Yaskawa INFORM job: aprem3TRJ1.JBI

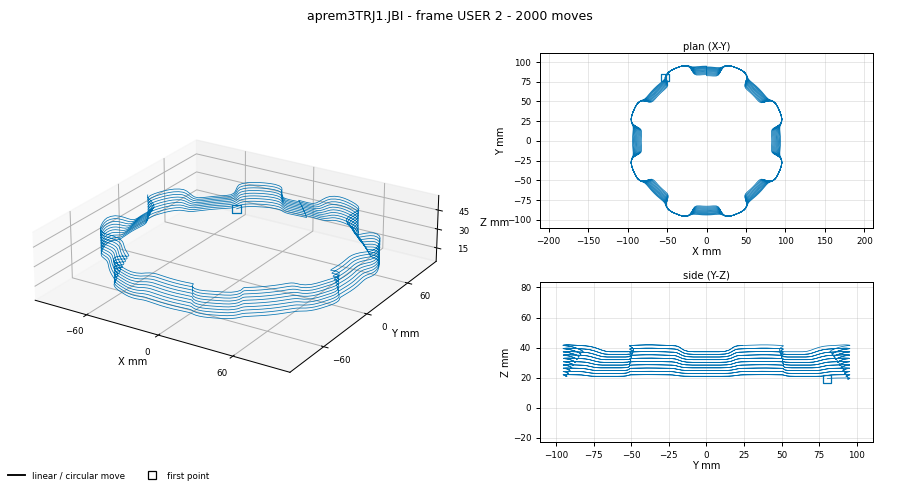
[picture p0: tool path of aprem3TRJ1.JBI in frame USER 2, 2000 of 2000 moves have a stored position in this frame; points joined in program order, loops and branches not executed]
/JOB
//NAME aprem3TRJ1
///FOLDERNAME DEMO
//POS
///NPOS 2000,0,2000,0,0,0
///USER 2
///TOOL 7
///POSTYPE USER
///RECTAN
///RCONF 1,0,0,0,0,0,0,0,0,0,0,0,0,0,0,0,0,0,0,0,0,0,0,0
C00000=-52.755,80.388,19.309,-171.7434,14.7955,-3566.7249
C00001=-51.961,81.931,19.493,-175.4363,10.0997,-3567.6170
C00002=-51.163,83.502,19.627,-176.4604,6.1368,-3568.5035
C00003=-49.917,85.194,19.692,-177.1673,3.1412,-3569.6330
C00004=-47.874,87.106,19.726,-178.6253,1.1228,-3571.2065
C00005=-45.272,88.975,19.753,-179.7684,0.1462,-3573.0322
C00006=-42.449,90.515,19.780,-179.9313,0.0331,-3574.8747
C00007=-39.659,91.796,19.798,-179.9923,0.0034,-3576.6340
C00008=-36.867,92.953,19.798,-179.9922,0.0031,-3578.3657
C00009=-33.988,94.020,19.780,-179.9280,0.0252,-3580.1252
C00010=-30.903,94.927,19.753,-179.7329,0.0604,-3581.9676
C00011=-27.741,95.446,19.726,-178.2343,0.1783,-3583.7937
C00012=-24.945,95.538,19.692,-175.7796,-0.2187,-3585.3667
C00013=-22.867,95.222,19.627,-173.1704,-1.8493,-3586.4965
C00014=-21.192,94.676,19.493,-169.6633,-3.9762,-3587.3831
C00015=-19.540,94.146,19.309,-163.8609,-4.8105,-3588.2747
C00016=-17.528,93.824,19.120,-157.6135,-2.4711,-3589.4181
C00017=-14.592,93.857,18.976,-154.0584,1.6115,-3591.1629
C00018=-10.190,94.262,18.917,-153.0799,2.7335,-3593.8301
C00019=-5.317,94.652,18.914,-152.9496,1.6756,-3596.7848
C00020=0.000,94.804,18.916,-152.9230,0.0002,-3600.0000
C00021=0.000,93.772,20.859,-151.1709,0.0003,-3600.0000
C00022=5.223,93.624,20.857,-151.1986,-1.7982,-3603.1930
C00023=10.031,93.243,20.860,-151.3318,-2.8339,-3606.1402
C00024=14.399,92.874,20.935,-152.4025,-1.1034,-3608.8129
C00025=17.292,92.935,21.118,-156.8210,4.1648,-3610.5402
C00026=19.271,93.399,21.361,-164.4264,6.3648,-3611.6582
C00027=20.902,94.108,21.598,-170.7334,4.7910,-3612.5225
C00028=22.556,94.852,21.773,-173.9772,2.3273,-3613.3766
C00029=24.607,95.353,21.858,-176.1452,0.4720,-3614.4702
C00030=27.423,95.407,21.902,-178.4246,-0.0969,-3616.0363
C00031=30.651,94.973,21.938,-179.8436,-0.0322,-3617.8866
C00032=33.828,94.073,21.973,-179.9356,-0.0223,-3619.7782
C00033=36.813,92.974,21.997,-179.9932,-0.0027,-3621.6011
C00034=39.712,91.773,21.997,-179.9933,-0.0029,-3623.3991
C00035=42.599,90.440,21.973,-179.9387,-0.0298,-3625.2213
C00036=45.483,88.829,21.938,-179.8667,-0.0878,-3627.1138
C00037=48.072,86.854,21.902,-178.8174,-1.0456,-3628.9637
C00038=50.025,84.825,21.858,-177.6053,-3.0607,-3630.5297
C00039=51.121,83.020,21.773,-177.3739,-5.9001,-3631.6234
C00040=51.765,81.324,21.598,-176.7889,-9.9060,-3632.4779
C00041=52.416,79.670,21.361,-173.2589,-15.4269,-3633.3415
C00042=53.488,77.942,21.118,-165.8953,-19.5067,-3634.4600
C00043=55.491,75.854,20.935,-159.0309,-19.5961,-3636.1873
C00044=58.840,73.026,20.860,-157.1386,-19.3725,-3638.8598
C00045=62.509,69.895,20.857,-157.6594,-20.1308,-3641.8071
C00046=66.307,66.307,20.859,-158.7340,-21.2663,-3645.0000
C00047=69.895,62.509,20.857,-159.8689,-22.3404,-3648.1929
C00048=73.026,58.840,20.860,-160.6271,-22.8610,-3651.1402
C00049=75.854,55.491,20.935,-160.4041,-20.9693,-3653.8127
C00050=77.942,53.488,21.118,-160.4933,-14.1047,-3655.5400
C00051=79.670,52.416,21.361,-164.5731,-6.7411,-3656.6585
C00052=81.324,51.765,21.598,-170.0940,-3.2111,-3657.5221
C00053=83.020,51.121,21.773,-174.0999,-2.6261,-3658.3766
C00054=84.825,50.025,21.858,-176.9393,-2.3947,-3659.4703
C00055=86.854,48.072,21.902,-178.9544,-1.1826,-3661.0363
C00056=88.829,45.483,21.938,-179.9122,-0.1333,-3662.8862
C00057=90.440,42.599,21.973,-179.9702,-0.0613,-3664.7787
C00058=91.773,39.712,21.997,-179.9971,-0.0067,-3666.6009
C00059=92.974,36.813,21.997,-179.9973,-0.0068,-3668.3989
C00060=94.073,33.828,21.973,-179.9777,-0.0644,-3670.2218
C00061=94.973,30.651,21.938,-179.9678,-0.1564,-3672.1134
C00062=95.407,27.423,21.902,-179.9031,-1.5754,-3673.9637
C00063=95.353,24.607,21.858,179.5280,-3.8548,-3675.5298
C00064=94.852,22.556,21.773,177.6727,-6.0228,-3676.6234
C00065=94.108,20.902,21.598,175.2090,-9.2666,-3677.4775
C00066=93.399,19.271,21.361,173.6352,-15.5736,-3678.3418
C00067=92.935,17.292,21.118,175.8352,-23.1790,-3679.4598
C00068=92.874,14.399,20.935,-178.8966,-27.5975,-3681.1871
C00069=93.243,10.031,20.860,-177.1661,-28.6682,-3683.8598
C00070=93.624,5.223,20.857,-178.2018,-28.8014,-3686.8070
C00071=93.772,0.000,20.859,179.9997,-28.8291,-3690.0000
C00072=93.624,-5.223,20.857,178.2021,-28.8014,-3693.1930
C00073=93.243,-10.031,20.860,177.1667,-28.6682,-3696.1402
C00074=92.875,-14.399,20.935,178.8963,-27.5974,-3698.8128
C00075=92.935,-17.292,21.118,-175.8352,-23.1790,-3700.5402
C00076=93.399,-19.271,21.361,-173.6352,-15.5736,-3701.6582
C00077=94.108,-20.902,21.598,-175.2090,-9.2666,-3702.5225
C00078=94.852,-22.556,21.773,-177.6727,-6.0228,-3703.3766
C00079=95.353,-24.607,21.858,-179.5280,-3.8548,-3704.4702
C00080=95.407,-27.423,21.902,179.9031,-1.5754,-3706.0363
C00081=94.973,-30.651,21.938,179.9678,-0.1564,-3707.8866
C00082=94.073,-33.828,21.973,179.9777,-0.0644,-3709.7782
C00083=92.974,-36.813,21.997,179.9973,-0.0068,-3711.6011
C00084=91.773,-39.712,21.997,179.9971,-0.0067,-3713.3991
C00085=90.440,-42.599,21.973,179.9702,-0.0613,-3715.2213
C00086=88.829,-45.483,21.938,179.9122,-0.1333,-3717.1138
C00087=86.854,-48.072,21.902,178.9544,-1.1826,-3718.9637
C00088=84.825,-50.025,21.858,176.9393,-2.3947,-3720.5297
C00089=83.020,-51.121,21.773,174.0999,-2.6261,-3721.6234
C00090=81.324,-51.765,21.598,170.0940,-3.2111,-3722.4779
C00091=79.670,-52.416,21.361,164.5731,-6.7411,-3723.3415
C00092=77.942,-53.488,21.118,160.4933,-14.1047,-3724.4600
C00093=75.854,-55.491,20.935,160.4039,-20.9691,-3726.1873
C00094=73.026,-58.840,20.860,160.6275,-22.8614,-3728.8598
C00095=69.895,-62.509,20.857,159.8692,-22.3406,-3731.8071
C00096=66.307,-66.307,20.859,158.7337,-21.2660,-3735.0000
C00097=62.509,-69.895,20.857,157.6596,-20.1311,-3738.1929
C00098=58.840,-73.026,20.860,157.1390,-19.3729,-3741.1402
C00099=55.491,-75.854,20.935,159.0307,-19.5959,-3743.8127
C00100=53.488,-77.942,21.118,165.8953,-19.5067,-3745.5400
C00101=52.416,-79.670,21.361,173.2589,-15.4269,-3746.6585
C00102=51.765,-81.324,21.598,176.7889,-9.9060,-3747.5221
C00103=51.121,-83.020,21.773,177.3739,-5.9001,-3748.3766
C00104=50.025,-84.825,21.858,177.6053,-3.0607,-3749.4703
C00105=48.072,-86.854,21.902,178.8174,-1.0456,-3751.0363
C00106=45.483,-88.829,21.938,179.8667,-0.0878,-3752.8862
C00107=42.599,-90.440,21.973,179.9387,-0.0298,-3754.7787
C00108=39.712,-91.773,21.997,179.9933,-0.0029,-3756.6009
C00109=36.813,-92.974,21.997,179.9932,-0.0027,-3758.3989
C00110=33.828,-94.073,21.973,179.9356,-0.0223,-3760.2218
C00111=30.651,-94.973,21.938,179.8436,-0.0322,-3762.1134
C00112=27.423,-95.407,21.902,178.4246,-0.0969,-3763.9637
C00113=24.607,-95.353,21.858,176.1452,0.4720,-3765.5298
C00114=22.556,-94.852,21.773,173.9772,2.3273,-3766.6234
C00115=20.902,-94.108,21.598,170.7334,4.7910,-3767.4775
C00116=19.271,-93.399,21.361,164.4264,6.3648,-3768.3418
C00117=17.292,-92.935,21.118,156.8210,4.1648,-3769.4598
C00118=14.399,-92.874,20.935,152.4025,-1.1034,-3771.1871
C00119=10.031,-93.243,20.860,151.3318,-2.8339,-3773.8598
C00120=5.223,-93.624,20.857,151.1986,-1.7982,-3776.8070
C00121=0.000,-93.772,20.859,151.1709,0.0003,-3780.0000
C00122=0.000,-93.772,20.859,151.1709,0.0003,-3780.0000
C00123=-5.223,-93.624,20.857,151.1986,1.7979,-3783.1930
C00124=-10.031,-93.243,20.860,151.3318,2.8333,-3786.1402
C00125=-14.399,-92.875,20.935,152.4026,1.1037,-3788.8128
C00126=-17.292,-92.935,21.118,156.8210,-4.1648,-3790.5402
C00127=-19.271,-93.399,21.361,164.4264,-6.3648,-3791.6582
C00128=-20.902,-94.108,21.598,170.7334,-4.7910,-3792.5225
C00129=-22.556,-94.852,21.773,173.9772,-2.3273,-3793.3766
C00130=-24.607,-95.353,21.858,176.1452,-0.4720,-3794.4702
C00131=-27.423,-95.407,21.902,178.4246,0.0969,-3796.0363
C00132=-30.651,-94.973,21.938,179.8436,0.0322,-3797.8866
C00133=-33.828,-94.073,21.973,179.9356,0.0223,-3799.7782
C00134=-36.813,-92.974,21.997,179.9932,0.0027,-3801.6011
C00135=-39.712,-91.773,21.997,179.9933,0.0029,-3803.3991
C00136=-42.599,-90.440,21.973,179.9387,0.0298,-3805.2213
C00137=-45.483,-88.829,21.938,179.8667,0.0878,-3807.1138
C00138=-48.072,-86.854,21.902,178.8174,1.0456,-3808.9637
C00139=-50.025,-84.825,21.858,177.6053,3.0607,-3810.5297
C00140=-51.121,-83.020,21.773,177.3739,5.9001,-3811.6234
C00141=-51.765,-81.324,21.598,176.7889,9.9060,-3812.4779
C00142=-52.416,-79.670,21.361,173.2589,15.4269,-3813.3415
C00143=-53.488,-77.942,21.118,165.8953,19.5067,-3814.4600
C00144=-55.491,-75.854,20.935,159.0309,19.5961,-3816.1873
C00145=-58.840,-73.026,20.860,157.1386,19.3725,-3818.8598
C00146=-62.509,-69.895,20.857,157.6594,20.1308,-3821.8071
C00147=-66.307,-66.307,20.859,158.7340,21.2663,-3825.0000
C00148=-69.895,-62.509,20.857,159.8689,22.3404,-3828.1929
C00149=-73.026,-58.840,20.860,160.6271,22.8610,-3831.1402
C00150=-75.854,-55.491,20.935,160.4041,20.9693,-3833.8127
C00151=-77.942,-53.488,21.118,160.4933,14.1047,-3835.5400
C00152=-79.670,-52.416,21.361,164.5731,6.7411,-3836.6585
C00153=-81.324,-51.765,21.598,170.0940,3.2111,-3837.5221
C00154=-83.020,-51.121,21.773,174.0999,2.6261,-3838.3766
C00155=-84.825,-50.025,21.858,176.9393,2.3947,-3839.4703
C00156=-86.854,-48.072,21.902,178.9544,1.1826,-3841.0363
C00157=-88.829,-45.483,21.938,179.9122,0.1333,-3842.8862
C00158=-90.440,-42.599,21.973,179.9702,0.0613,-3844.7787
C00159=-91.773,-39.712,21.997,179.9971,0.0067,-3846.6009
C00160=-92.974,-36.813,21.997,179.9973,0.0068,-3848.3989
C00161=-94.073,-33.828,21.973,179.9777,0.0644,-3850.2218
C00162=-94.973,-30.651,21.938,179.9678,0.1564,-3852.1134
C00163=-95.407,-27.423,21.902,179.9031,1.5754,-3853.9637
C00164=-95.353,-24.607,21.858,-179.5280,3.8548,-3855.5298
C00165=-94.852,-22.556,21.773,-177.6727,6.0228,-3856.6234
C00166=-94.108,-20.902,21.598,-175.2090,9.2666,-3857.4775
C00167=-93.399,-19.271,21.361,-173.6352,15.5736,-3858.3418
C00168=-92.935,-17.292,21.118,-175.8352,23.1790,-3859.4598
C00169=-92.874,-14.399,20.935,178.8966,27.5975,-3861.1871
C00170=-93.243,-10.031,20.860,177.1661,28.6682,-3863.8598
C00171=-93.624,-5.223,20.857,178.2018,28.8014,-3866.8070
C00172=-93.772,0.000,20.859,-179.9997,28.8291,-3870.0000
C00173=-93.624,5.223,20.857,-178.2021,28.8014,-3873.1930
C00174=-93.243,10.031,20.860,-177.1667,28.6682,-3876.1402
C00175=-92.875,14.399,20.935,-178.8963,27.5974,-3878.8128
C00176=-92.935,17.292,21.118,175.8352,23.1790,-3880.5402
C00177=-93.399,19.271,21.361,173.6352,15.5736,-3881.6582
C00178=-94.108,20.902,21.598,175.2090,9.2666,-3882.5225
C00179=-94.852,22.556,21.773,177.6727,6.0228,-3883.3766
C00180=-95.353,24.607,21.858,179.5280,3.8548,-3884.4702
C00181=-95.407,27.423,21.902,-179.9031,1.5754,-3886.0363
C00182=-94.973,30.651,21.938,-179.9678,0.1564,-3887.8866
C00183=-94.073,33.828,21.973,-179.9777,0.0644,-3889.7782
C00184=-92.974,36.813,21.997,-179.9973,0.0068,-3891.6011
C00185=-91.773,39.712,21.997,-179.9971,0.0067,-3893.3991
C00186=-90.440,42.599,21.973,-179.9702,0.0613,-3895.2213
C00187=-88.829,45.483,21.938,-179.9122,0.1333,-3897.1138
C00188=-86.854,48.072,21.902,-178.9544,1.1826,-3898.9637
C00189=-84.825,50.025,21.858,-176.9393,2.3947,-3900.5297
C00190=-83.020,51.121,21.773,-174.0999,2.6261,-3901.6234
C00191=-81.324,51.765,21.598,-170.0940,3.2111,-3902.4779
C00192=-79.670,52.416,21.361,-164.5731,6.7411,-3903.3415
C00193=-77.942,53.488,21.118,-160.4933,14.1047,-3904.4600
C00194=-75.854,55.491,20.935,-160.4039,20.9691,-3906.1873
C00195=-73.026,58.840,20.860,-160.6275,22.8614,-3908.8598
C00196=-69.895,62.509,20.857,-159.8692,22.3406,-3911.8071
C00197=-66.307,66.307,20.859,-158.7337,21.2660,-3915.0000
C00198=-62.509,69.895,20.857,-157.6596,20.1311,-3918.1929
C00199=-58.840,73.026,20.860,-157.1390,19.3729,-3921.1402
C00200=-55.491,75.854,20.935,-159.0307,19.5959,-3923.8127
C00201=-53.488,77.942,21.118,-165.8953,19.5067,-3925.5400
C00202=-52.416,79.670,21.361,-173.2589,15.4269,-3926.6585
C00203=-51.765,81.324,21.598,-176.7889,9.9060,-3927.5221
C00204=-51.121,83.020,21.773,-177.3739,5.9001,-3928.3766
C00205=-50.025,84.825,21.858,-177.6053,3.0607,-3929.4703
C00206=-48.072,86.854,21.902,-178.8174,1.0456,-3931.0363
C00207=-45.483,88.829,21.938,-179.8667,0.0878,-3932.8862
C00208=-42.599,90.440,21.973,-179.9387,0.0298,-3934.7787
C00209=-39.712,91.773,21.997,-179.9933,0.0029,-3936.6009
C00210=-36.813,92.974,21.997,-179.9932,0.0027,-3938.3989
C00211=-33.828,94.073,21.973,-179.9356,0.0223,-3940.2218
C00212=-30.651,94.973,21.938,-179.8436,0.0322,-3942.1134
C00213=-27.423,95.407,21.902,-178.4246,0.0969,-3943.9637
C00214=-24.607,95.353,21.858,-176.1452,-0.4720,-3945.5298
C00215=-22.556,94.852,21.773,-173.9772,-2.3273,-3946.6234
C00216=-20.902,94.108,21.598,-170.7334,-4.7910,-3947.4775
C00217=-19.271,93.399,21.361,-164.4264,-6.3648,-3948.3418
C00218=-17.292,92.935,21.118,-156.8210,-4.1648,-3949.4598
C00219=-14.399,92.875,20.935,-152.4026,1.1037,-3951.1872
C00220=-10.031,93.243,20.860,-151.3318,2.8333,-3953.8598
C00221=-5.223,93.624,20.857,-151.1986,1.7979,-3956.8070
C00222=0.000,93.772,20.859,-151.1709,0.0003,-3960.0000
C00223=0.000,92.684,22.771,-149.6099,0.0003,-3960.0000
C00224=5.124,92.540,22.769,-149.6384,-1.9089,-3963.1693
C00225=9.864,92.169,22.773,-149.7740,-2.8935,-3966.1086
C00226=14.194,91.838,22.865,-150.9609,-0.4562,-3968.7858
C00227=17.042,91.994,23.091,-156.4950,5.9927,-3970.4951
C00228=18.986,92.606,23.393,-165.5257,7.6266,-3971.5862
C00229=20.592,93.503,23.691,-172.1237,5.1935,-3972.4199
C00230=22.223,94.456,23.912,-175.0607,2.5303,-3973.2394
C00231=24.245,95.156,24.019,-176.7061,0.6541,-3974.2944
C00232=27.082,95.366,24.075,-178.6926,-0.0269,-3975.8535
C00233=30.380,95.022,24.120,-179.9786,-0.0040,-3977.7299
C00234=33.658,94.129,24.166,-179.9455,-0.0187,-3979.6757
C00235=36.755,92.996,24.196,-179.9945,-0.0022,-3981.5655
C00236=39.769,91.748,24.196,-179.9946,-0.0024,-3983.4348
C00237=42.760,90.359,24.166,-179.9482,-0.0253,-3985.3246
C00238=45.709,88.673,24.120,-179.9821,-0.0123,-3987.2701
C00239=48.284,86.584,24.075,-179.0565,-0.9056,-3989.1464
C00240=50.142,84.429,24.019,-178.1315,-2.7920,-3990.7059
C00241=51.076,82.504,23.912,-178.2896,-5.2767,-3991.7605
C00242=51.556,80.678,23.691,-178.0785,-9.2071,-3992.5800
C00243=52.057,78.907,23.393,-174.9794,-15.4942,-3993.4139
C00244=52.999,77.101,23.091,-166.8676,-20.8949,-3994.5045
C00245=54.903,74.976,22.865,-158.2868,-21.1542,-3996.2144
C00246=58.198,72.148,22.773,-155.8812,-20.6181,-3998.8913
C00247=61.813,69.059,22.769,-156.3569,-21.3383,-4001.8309
C00248=65.538,65.538,22.771,-157.4767,-22.5237,-4005.0000
C00249=69.059,61.813,22.769,-158.6615,-23.6429,-4008.1691
C00250=72.148,58.198,22.773,-159.3815,-24.1184,-4011.1087
C00251=74.976,54.903,22.865,-158.8460,-21.7135,-4013.7856
C00252=77.101,52.999,23.091,-159.1051,-13.1324,-4015.4955
C00253=78.907,52.057,23.393,-164.5058,-5.0206,-4016.5861
C00254=80.678,51.556,23.691,-170.7929,-1.9215,-4017.4200
C00255=82.504,51.076,23.912,-174.7233,-1.7104,-4018.2395
C00256=84.429,50.142,24.019,-177.2080,-1.8685,-4019.2941
C00257=86.584,48.284,24.075,-179.0944,-0.9435,-4020.8536
C00258=88.673,45.709,24.120,-179.9877,-0.0179,-4022.7299
C00259=90.359,42.760,24.166,-179.9747,-0.0518,-4024.6754
C00260=91.748,39.769,24.196,-179.9976,-0.0054,-4026.5652
C00261=92.996,36.755,24.196,-179.9978,-0.0055,-4028.4345
C00262=94.129,33.658,24.166,-179.9813,-0.0545,-4030.3243
C00263=95.022,30.380,24.120,-179.9960,-0.0214,-4032.2701
C00264=95.366,27.082,24.075,-179.9731,-1.3074,-4034.1465
C00265=95.156,24.245,24.019,179.3459,-3.2939,-4035.7056
C00266=94.456,22.223,23.912,177.4697,-4.9393,-4036.7606
C00267=93.503,20.592,23.691,174.8065,-7.8763,-4037.5801
C00268=92.606,18.986,23.393,172.3734,-14.4743,-4038.4138
C00269=91.994,17.042,23.091,174.0073,-23.5050,-4039.5049
C00270=91.838,14.194,22.865,-179.5438,-29.0391,-4041.2142
C00271=92.169,9.864,22.773,-177.1065,-30.2260,-4043.8914
C00272=92.540,5.124,22.769,-178.0911,-30.3616,-4046.8307
C00273=92.684,0.000,22.771,179.9997,-30.3901,-4050.0000
C00274=92.540,-5.124,22.769,178.0916,-30.3616,-4053.1693
C00275=92.169,-9.864,22.773,177.1071,-30.2260,-4056.1086
C00276=91.838,-14.194,22.865,179.5434,-29.0390,-4058.7858
C00277=91.994,-17.042,23.091,-174.0073,-23.5050,-4060.4951
C00278=92.606,-18.986,23.393,-172.3734,-14.4743,-4061.5862
C00279=93.503,-20.592,23.691,-174.8065,-7.8763,-4062.4199
C00280=94.456,-22.223,23.912,-177.4697,-4.9393,-4063.2394
C00281=95.156,-24.245,24.019,-179.3459,-3.2939,-4064.2944
C00282=95.366,-27.082,24.075,179.9731,-1.3074,-4065.8535
C00283=95.022,-30.380,24.120,179.9960,-0.0214,-4067.7299
C00284=94.129,-33.658,24.166,179.9813,-0.0545,-4069.6757
C00285=92.996,-36.755,24.196,179.9978,-0.0055,-4071.5655
C00286=91.748,-39.769,24.196,179.9976,-0.0054,-4073.4348
C00287=90.359,-42.760,24.166,179.9747,-0.0518,-4075.3246
C00288=88.673,-45.709,24.120,179.9877,-0.0179,-4077.2701
C00289=86.584,-48.284,24.075,179.0944,-0.9435,-4079.1464
C00290=84.429,-50.142,24.019,177.2080,-1.8685,-4080.7059
C00291=82.504,-51.076,23.912,174.7233,-1.7104,-4081.7605
C00292=80.678,-51.556,23.691,170.7929,-1.9215,-4082.5800
C00293=78.907,-52.057,23.393,164.5058,-5.0206,-4083.4139
C00294=77.101,-52.999,23.091,159.1051,-13.1324,-4084.5045
C00295=74.976,-54.903,22.865,158.8458,-21.7132,-4086.2144
C00296=72.148,-58.198,22.773,159.3819,-24.1188,-4088.8913
C00297=69.059,-61.813,22.769,158.6617,-23.6431,-4091.8309
C00298=65.538,-65.538,22.771,157.4763,-22.5233,-4095.0000
C00299=61.813,-69.059,22.769,156.3571,-21.3385,-4098.1691
C00300=58.198,-72.148,22.773,155.8816,-20.6185,-4101.1087
C00301=54.903,-74.976,22.865,158.2865,-21.1540,-4103.7856
C00302=52.999,-77.101,23.091,166.8676,-20.8949,-4105.4955
C00303=52.057,-78.907,23.393,174.9794,-15.4942,-4106.5861
C00304=51.556,-80.678,23.691,178.0785,-9.2071,-4107.4200
C00305=51.076,-82.504,23.912,178.2896,-5.2767,-4108.2395
C00306=50.142,-84.429,24.019,178.1315,-2.7920,-4109.2941
C00307=48.284,-86.584,24.075,179.0565,-0.9056,-4110.8536
C00308=45.709,-88.673,24.120,179.9821,-0.0123,-4112.7299
C00309=42.760,-90.359,24.166,179.9482,-0.0253,-4114.6754
C00310=39.769,-91.748,24.196,179.9946,-0.0024,-4116.5652
C00311=36.755,-92.996,24.196,179.9945,-0.0022,-4118.4345
C00312=33.658,-94.129,24.166,179.9455,-0.0187,-4120.3243
C00313=30.380,-95.022,24.120,179.9786,-0.0040,-4122.2701
C00314=27.082,-95.366,24.075,178.6926,-0.0269,-4124.1465
C00315=24.245,-95.156,24.019,176.7061,0.6541,-4125.7056
C00316=22.223,-94.456,23.912,175.0607,2.5303,-4126.7606
C00317=20.592,-93.503,23.691,172.1237,5.1935,-4127.5801
C00318=18.986,-92.606,23.393,165.5257,7.6266,-4128.4138
C00319=17.042,-91.994,23.091,156.4950,5.9927,-4129.5049
C00320=14.194,-91.838,22.865,150.9609,-0.4562,-4131.2142
C00321=9.864,-92.169,22.773,149.7740,-2.8935,-4133.8914
C00322=5.124,-92.540,22.769,149.6384,-1.9089,-4136.8307
C00323=0.000,-92.684,22.771,149.6099,0.0003,-4140.0000
C00324=0.000,-92.684,22.771,149.6099,0.0003,-4140.0000
C00325=-5.124,-92.540,22.769,149.6384,1.9084,-4143.1693
C00326=-9.864,-92.169,22.773,149.7740,2.8929,-4146.1086
C00327=-14.194,-91.838,22.865,150.9610,0.4566,-4148.7858
C00328=-17.042,-91.994,23.091,156.4950,-5.9927,-4150.4951
C00329=-18.986,-92.606,23.393,165.5257,-7.6266,-4151.5862
C00330=-20.592,-93.503,23.691,172.1237,-5.1935,-4152.4199
C00331=-22.223,-94.456,23.912,175.0607,-2.5303,-4153.2394
C00332=-24.245,-95.156,24.019,176.7061,-0.6541,-4154.2944
C00333=-27.082,-95.366,24.075,178.6926,0.0269,-4155.8535
C00334=-30.380,-95.022,24.120,179.9786,0.0040,-4157.7299
C00335=-33.658,-94.129,24.166,179.9455,0.0187,-4159.6757
C00336=-36.755,-92.996,24.196,179.9945,0.0022,-4161.5655
C00337=-39.769,-91.748,24.196,179.9946,0.0024,-4163.4348
C00338=-42.760,-90.359,24.166,179.9482,0.0253,-4165.3246
C00339=-45.709,-88.673,24.120,179.9821,0.0123,-4167.2701
C00340=-48.284,-86.584,24.075,179.0565,0.9056,-4169.1464
C00341=-50.142,-84.429,24.019,178.1315,2.7920,-4170.7059
C00342=-51.076,-82.504,23.912,178.2896,5.2767,-4171.7605
C00343=-51.556,-80.678,23.691,178.0785,9.2071,-4172.5800
C00344=-52.057,-78.907,23.393,174.9794,15.4942,-4173.4139
C00345=-52.999,-77.101,23.091,166.8676,20.8949,-4174.5045
C00346=-54.903,-74.976,22.865,158.2868,21.1542,-4176.2144
C00347=-58.198,-72.148,22.773,155.8812,20.6181,-4178.8913
C00348=-61.813,-69.059,22.769,156.3569,21.3383,-4181.8309
C00349=-65.538,-65.538,22.771,157.4767,22.5237,-4185.0000
C00350=-69.059,-61.813,22.769,158.6615,23.6429,-4188.1691
C00351=-72.148,-58.198,22.773,159.3815,24.1184,-4191.1087
C00352=-74.976,-54.903,22.865,158.8460,21.7135,-4193.7856
C00353=-77.101,-52.999,23.091,159.1051,13.1324,-4195.4955
C00354=-78.907,-52.057,23.393,164.5058,5.0206,-4196.5861
C00355=-80.678,-51.556,23.691,170.7929,1.9215,-4197.4200
C00356=-82.504,-51.076,23.912,174.7233,1.7104,-4198.2395
C00357=-84.429,-50.142,24.019,177.2080,1.8685,-4199.2941
C00358=-86.584,-48.284,24.075,179.0944,0.9435,-4200.8536
C00359=-88.673,-45.709,24.120,179.9877,0.0179,-4202.7299
C00360=-90.359,-42.760,24.166,179.9747,0.0518,-4204.6754
C00361=-91.748,-39.769,24.196,179.9976,0.0054,-4206.5652
C00362=-92.996,-36.755,24.196,179.9978,0.0055,-4208.4345
C00363=-94.129,-33.658,24.166,179.9813,0.0545,-4210.3243
C00364=-95.022,-30.380,24.120,179.9960,0.0214,-4212.2701
C00365=-95.366,-27.082,24.075,179.9731,1.3074,-4214.1465
C00366=-95.156,-24.245,24.019,-179.3459,3.2939,-4215.7056
C00367=-94.456,-22.223,23.912,-177.4697,4.9393,-4216.7606
C00368=-93.503,-20.592,23.691,-174.8065,7.8763,-4217.5801
C00369=-92.606,-18.986,23.393,-172.3734,14.4743,-4218.4138
C00370=-91.994,-17.042,23.091,-174.0073,23.5050,-4219.5049
C00371=-91.838,-14.194,22.865,179.5438,29.0391,-4221.2142
C00372=-92.169,-9.864,22.773,177.1065,30.2260,-4223.8914
C00373=-92.540,-5.124,22.769,178.0911,30.3616,-4226.8307
C00374=-92.684,0.000,22.771,-179.9997,30.3901,-4230.0000
C00375=-92.540,5.124,22.769,-178.0916,30.3616,-4233.1693
C00376=-92.169,9.864,22.773,-177.1071,30.2260,-4236.1086
C00377=-91.838,14.194,22.865,-179.5434,29.0390,-4238.7858
C00378=-91.994,17.042,23.091,174.0073,23.5050,-4240.4951
C00379=-92.606,18.986,23.393,172.3734,14.4743,-4241.5862
C00380=-93.503,20.592,23.691,174.8065,7.8763,-4242.4199
C00381=-94.456,22.223,23.912,177.4697,4.9393,-4243.2394
C00382=-95.156,24.245,24.019,179.3459,3.2939,-4244.2944
C00383=-95.366,27.082,24.075,-179.9731,1.3074,-4245.8535
C00384=-95.022,30.380,24.120,-179.9960,0.0214,-4247.7299
C00385=-94.129,33.658,24.166,-179.9813,0.0545,-4249.6757
C00386=-92.996,36.755,24.196,-179.9978,0.0055,-4251.5655
C00387=-91.748,39.769,24.196,-179.9976,0.0054,-4253.4348
C00388=-90.359,42.760,24.166,-179.9747,0.0518,-4255.3246
C00389=-88.673,45.709,24.120,-179.9877,0.0179,-4257.2701
C00390=-86.584,48.284,24.075,-179.0944,0.9435,-4259.1464
C00391=-84.429,50.142,24.019,-177.2080,1.8685,-4260.7059
C00392=-82.504,51.076,23.912,-174.7233,1.7104,-4261.7605
C00393=-80.678,51.556,23.691,-170.7929,1.9215,-4262.5800
C00394=-78.907,52.057,23.393,-164.5058,5.0206,-4263.4139
C00395=-77.101,52.999,23.091,-159.1051,13.1324,-4264.5045
C00396=-74.976,54.903,22.865,-158.8458,21.7132,-4266.2144
C00397=-72.148,58.198,22.773,-159.3819,24.1188,-4268.8913
C00398=-69.059,61.813,22.769,-158.6617,23.6431,-4271.8309
C00399=-65.538,65.538,22.771,-157.4763,22.5233,-4275.0000
C00400=-61.813,69.059,22.769,-156.3571,21.3385,-4278.1691
C00401=-58.198,72.148,22.773,-155.8816,20.6185,-4281.1087
C00402=-54.903,74.976,22.865,-158.2865,21.1540,-4283.7856
C00403=-52.999,77.101,23.091,-166.8676,20.8949,-4285.4955
C00404=-52.057,78.907,23.393,-174.9794,15.4942,-4286.5861
C00405=-51.556,80.678,23.691,-178.0785,9.2071,-4287.4200
C00406=-51.076,82.504,23.912,-178.2896,5.2767,-4288.2395
C00407=-50.142,84.429,24.019,-178.1315,2.7920,-4289.2941
C00408=-48.284,86.584,24.075,-179.0565,0.9056,-4290.8536
C00409=-45.709,88.673,24.120,-179.9821,0.0123,-4292.7299
C00410=-42.760,90.359,24.166,-179.9482,0.0253,-4294.6754
C00411=-39.769,91.748,24.196,-179.9946,0.0024,-4296.5652
C00412=-36.755,92.996,24.196,-179.9945,0.0022,-4298.4345
C00413=-33.658,94.129,24.166,-179.9455,0.0187,-4300.3243
C00414=-30.380,95.022,24.120,-179.9786,0.0040,-4302.2701
C00415=-27.082,95.366,24.075,-178.6926,0.0269,-4304.1465
C00416=-24.245,95.156,24.019,-176.7061,-0.6541,-4305.7056
C00417=-22.223,94.456,23.912,-175.0607,-2.5303,-4306.7606
C00418=-20.592,93.503,23.691,-172.1237,-5.1935,-4307.5801
C00419=-18.986,92.606,23.393,-165.5257,-7.6266,-4308.4138
C00420=-17.042,91.994,23.091,-156.4950,-5.9927,-4309.5049
C00421=-14.194,91.838,22.865,-150.9610,0.4566,-4311.2142
C00422=-9.864,92.169,22.773,-149.7740,2.8929,-4313.8914
C00423=-5.124,92.540,22.769,-149.6384,1.9084,-4316.8307
C00424=0.000,92.684,22.771,-149.6099,0.0003,-4320.0000
C00425=0.000,91.548,24.655,-148.2220,0.0004,-4320.0000
C00426=5.020,91.408,24.652,-148.2512,-2.0082,-4323.1434
C00427=9.690,91.047,24.657,-148.3888,-2.9141,-4326.0750
C00428=13.981,90.755,24.767,-149.7234,0.3213,-4328.7577
C00429=16.781,91.008,25.041,-156.6468,7.8344,-4330.4474
C00430=18.686,91.772,25.406,-167.0189,8.4697,-4331.5089
C00431=20.265,92.865,25.771,-173.6442,5.1590,-4332.3101
C00432=21.871,94.037,26.043,-176.2884,2.4064,-4333.0930
C00433=23.861,94.948,26.175,-177.4309,0.7190,-4334.1066
C00434=26.720,95.323,26.245,-179.0289,0.0208,-4335.6587
C00435=30.093,95.074,26.301,179.8658,0.0220,-4337.5637
C00436=33.476,94.189,26.358,-179.9573,-0.0145,-4339.5659
C00437=36.693,93.020,26.395,-179.9960,-0.0016,-4341.5274
C00438=39.829,91.721,26.395,-179.9960,-0.0018,-4343.4725
C00439=42.931,90.273,26.358,-179.9596,-0.0199,-4345.4343
C00440=45.948,88.507,26.301,179.8895,0.0793,-4347.4359
C00441=48.509,86.297,26.245,-179.3280,-0.7014,-4349.3411
C00442=50.266,84.010,26.175,-178.6908,-2.3250,-4350.8935
C00443=51.029,81.959,26.043,-179.0745,-4.3225,-4351.9071
C00444=51.336,79.995,25.771,-179.1451,-8.1159,-4352.6899
C00445=51.679,78.105,25.406,-176.6973,-15.0186,-4353.4910
C00446=52.487,76.218,25.041,-168.2493,-21.9298,-4354.5530
C00447=54.287,74.059,24.767,-157.7629,-22.6253,-4356.2423
C00448=57.528,71.231,24.657,-154.7702,-21.7624,-4358.9252
C00449=61.085,68.184,24.652,-155.1868,-22.4287,-4361.8567
C00450=64.734,64.734,24.655,-156.3444,-23.6560,-4365.0000
C00451=68.184,61.085,24.652,-157.5710,-24.8129,-4368.1433
C00452=71.231,57.528,24.657,-158.2372,-25.2293,-4371.0748
C00453=74.059,54.287,24.767,-157.3750,-22.2374,-4373.7577
C00454=76.218,52.487,25.041,-158.0702,-11.7507,-4375.4470
C00455=78.105,51.679,25.406,-164.9814,-3.3027,-4376.5090
C00456=79.995,51.336,25.771,-171.8841,-0.8549,-4377.3101
C00457=81.959,51.029,26.043,-175.6775,-0.9255,-4378.0929
C00458=84.010,50.266,26.175,-177.6750,-1.3092,-4379.1065
C00459=86.297,48.509,26.245,-179.2986,-0.6720,-4380.6589
C00460=88.507,45.948,26.301,179.9207,0.1105,-4382.5641
C00461=90.273,42.931,26.358,-179.9801,-0.0404,-4384.5657
C00462=91.721,39.829,26.395,-179.9982,-0.0040,-4386.5275
C00463=93.020,36.693,26.395,-179.9984,-0.0040,-4388.4726
C00464=94.189,33.476,26.358,-179.9855,-0.0427,-4390.4341
C00465=95.074,30.093,26.301,179.9780,0.1342,-4392.4363
C00466=95.323,26.720,26.245,179.9792,-0.9711,-4394.3413
C00467=94.948,23.861,26.175,179.2810,-2.5691,-4395.8934
C00468=94.037,21.871,26.043,177.5936,-3.7116,-4396.9070
C00469=92.865,20.265,25.771,174.8410,-6.3558,-4397.6899
C00470=91.772,18.686,25.406,171.5303,-12.9811,-4398.4911
C00471=91.008,16.781,25.041,172.1656,-23.3532,-4399.5526
C00472=90.755,13.981,24.767,179.6787,-30.2766,-4401.2423
C00473=91.047,9.690,24.657,-177.0859,-31.6112,-4403.9250
C00474=91.408,5.020,24.652,-177.9918,-31.7488,-4406.8566
C00475=91.548,0.000,24.655,179.9996,-31.7780,-4410.0000
C00476=91.408,-5.020,24.652,177.9923,-31.7488,-4413.1434
C00477=91.047,-9.690,24.657,177.0867,-31.6111,-4416.0750
C00478=90.755,-13.981,24.767,-179.6793,-30.2766,-4418.7577
C00479=91.008,-16.781,25.041,-172.1656,-23.3532,-4420.4474
C00480=91.772,-18.686,25.406,-171.5303,-12.9811,-4421.5089
C00481=92.865,-20.265,25.771,-174.8410,-6.3558,-4422.3101
C00482=94.037,-21.871,26.043,-177.5936,-3.7116,-4423.0930
C00483=94.948,-23.861,26.175,-179.2810,-2.5691,-4424.1066
C00484=95.323,-26.720,26.245,-179.9792,-0.9711,-4425.6587
C00485=95.074,-30.093,26.301,-179.9780,0.1342,-4427.5637
C00486=94.189,-33.476,26.358,179.9855,-0.0427,-4429.5659
C00487=93.020,-36.693,26.395,179.9984,-0.0040,-4431.5274
C00488=91.721,-39.829,26.395,179.9982,-0.0040,-4433.4725
C00489=90.273,-42.931,26.358,179.9801,-0.0404,-4435.4343
C00490=88.507,-45.948,26.301,-179.9207,0.1105,-4437.4359
C00491=86.297,-48.509,26.245,179.2986,-0.6720,-4439.3411
C00492=84.010,-50.266,26.175,177.6750,-1.3092,-4440.8935
C00493=81.959,-51.029,26.043,175.6775,-0.9255,-4441.9071
C00494=79.995,-51.336,25.771,171.8841,-0.8549,-4442.6899
C00495=78.105,-51.679,25.406,164.9814,-3.3027,-4443.4910
C00496=76.218,-52.487,25.041,158.0702,-11.7507,-4444.5530
C00497=74.059,-54.287,24.767,157.3747,-22.2371,-4446.2423
C00498=71.231,-57.528,24.657,158.2376,-25.2298,-4448.9252
C00499=68.184,-61.085,24.652,157.5713,-24.8132,-4451.8567
C00500=64.734,-64.734,24.655,156.3440,-23.6556,-4455.0000
C00501=61.085,-68.184,24.652,155.1871,-22.4290,-4458.1433
C00502=57.528,-71.231,24.657,154.7707,-21.7628,-4461.0748
C00503=54.287,-74.059,24.767,157.7626,-22.6250,-4463.7577
C00504=52.487,-76.218,25.041,168.2493,-21.9298,-4465.4470
C00505=51.679,-78.105,25.406,176.6973,-15.0186,-4466.5090
C00506=51.336,-79.995,25.771,179.1451,-8.1159,-4467.3101
C00507=51.029,-81.959,26.043,179.0745,-4.3225,-4468.0929
C00508=50.266,-84.010,26.175,178.6908,-2.3250,-4469.1065
C00509=48.509,-86.297,26.245,179.3280,-0.7014,-4470.6589
C00510=45.948,-88.507,26.301,-179.8895,0.0793,-4472.5641
C00511=42.931,-90.273,26.358,179.9596,-0.0199,-4474.5657
C00512=39.829,-91.721,26.395,179.9960,-0.0018,-4476.5275
C00513=36.693,-93.020,26.395,179.9960,-0.0016,-4478.4726
C00514=33.476,-94.189,26.358,179.9573,-0.0145,-4480.4341
C00515=30.093,-95.074,26.301,-179.8658,0.0220,-4482.4363
C00516=26.720,-95.323,26.245,179.0289,0.0208,-4484.3413
C00517=23.861,-94.948,26.175,177.4309,0.7190,-4485.8934
C00518=21.871,-94.037,26.043,176.2884,2.4064,-4486.9070
C00519=20.265,-92.865,25.771,173.6442,5.1590,-4487.6899
C00520=18.686,-91.772,25.406,167.0189,8.4697,-4488.4911
C00521=16.781,-91.008,25.041,156.6468,7.8344,-4489.5526
C00522=13.981,-90.755,24.767,149.7234,0.3213,-4491.2423
C00523=9.690,-91.047,24.657,148.3888,-2.9141,-4493.9250
C00524=5.020,-91.408,24.652,148.2512,-2.0082,-4496.8566
C00525=0.000,-91.548,24.655,148.2220,0.0004,-4500.0000
C00526=0.000,-91.548,24.655,148.2220,0.0004,-4500.0000
C00527=-5.020,-91.408,24.652,148.2512,2.0077,-4503.1434
C00528=-9.690,-91.047,24.657,148.3889,2.9133,-4506.0750
C00529=-13.981,-90.755,24.767,149.7234,-0.3207,-4508.7577
C00530=-16.781,-91.008,25.041,156.6468,-7.8344,-4510.4474
C00531=-18.686,-91.772,25.406,167.0189,-8.4697,-4511.5089
C00532=-20.265,-92.865,25.771,173.6442,-5.1590,-4512.3101
C00533=-21.871,-94.037,26.043,176.2884,-2.4064,-4513.0930
C00534=-23.861,-94.948,26.175,177.4309,-0.7190,-4514.1066
C00535=-26.720,-95.323,26.245,179.0289,-0.0208,-4515.6587
C00536=-30.093,-95.074,26.301,-179.8658,-0.0220,-4517.5637
C00537=-33.476,-94.189,26.358,179.9573,0.0145,-4519.5659
C00538=-36.693,-93.020,26.395,179.9960,0.0016,-4521.5274
C00539=-39.829,-91.721,26.395,179.9960,0.0018,-4523.4725
C00540=-42.931,-90.273,26.358,179.9596,0.0199,-4525.4343
C00541=-45.948,-88.507,26.301,-179.8895,-0.0793,-4527.4359
C00542=-48.509,-86.297,26.245,179.3280,0.7014,-4529.3411
C00543=-50.266,-84.010,26.175,178.6908,2.3250,-4530.8935
C00544=-51.029,-81.959,26.043,179.0745,4.3225,-4531.9071
C00545=-51.336,-79.995,25.771,179.1451,8.1159,-4532.6899
C00546=-51.679,-78.105,25.406,176.6973,15.0186,-4533.4910
C00547=-52.487,-76.218,25.041,168.2493,21.9298,-4534.5530
C00548=-54.287,-74.059,24.767,157.7629,22.6253,-4536.2423
C00549=-57.528,-71.231,24.657,154.7702,21.7624,-4538.9252
C00550=-61.085,-68.184,24.652,155.1868,22.4287,-4541.8567
C00551=-64.734,-64.734,24.655,156.3444,23.6560,-4545.0000
C00552=-68.184,-61.085,24.652,157.5710,24.8129,-4548.1433
C00553=-71.231,-57.528,24.657,158.2372,25.2293,-4551.0748
C00554=-74.059,-54.287,24.767,157.3750,22.2374,-4553.7577
C00555=-76.218,-52.487,25.041,158.0702,11.7507,-4555.4470
C00556=-78.105,-51.679,25.406,164.9814,3.3027,-4556.5090
C00557=-79.995,-51.336,25.771,171.8841,0.8549,-4557.3101
C00558=-81.959,-51.029,26.043,175.6775,0.9255,-4558.0929
C00559=-84.010,-50.266,26.175,177.6750,1.3092,-4559.1065
C00560=-86.297,-48.509,26.245,179.2986,0.6720,-4560.6589
C00561=-88.507,-45.948,26.301,-179.9207,-0.1105,-4562.5641
C00562=-90.273,-42.931,26.358,179.9801,0.0404,-4564.5657
C00563=-91.721,-39.829,26.395,179.9982,0.0040,-4566.5275
C00564=-93.020,-36.693,26.395,179.9984,0.0040,-4568.4726
C00565=-94.189,-33.476,26.358,179.9855,0.0427,-4570.4341
C00566=-95.074,-30.093,26.301,-179.9780,-0.1342,-4572.4363
C00567=-95.323,-26.720,26.245,-179.9792,0.9711,-4574.3413
C00568=-94.948,-23.861,26.175,-179.2810,2.5691,-4575.8934
C00569=-94.037,-21.871,26.043,-177.5936,3.7116,-4576.9070
C00570=-92.865,-20.265,25.771,-174.8410,6.3558,-4577.6899
C00571=-91.772,-18.686,25.406,-171.5303,12.9811,-4578.4911
C00572=-91.008,-16.781,25.041,-172.1656,23.3532,-4579.5526
C00573=-90.755,-13.981,24.767,-179.6787,30.2766,-4581.2423
C00574=-91.047,-9.690,24.657,177.0859,31.6112,-4583.9250
C00575=-91.408,-5.020,24.652,177.9918,31.7488,-4586.8566
C00576=-91.548,0.000,24.655,-179.9996,31.7780,-4590.0000
C00577=-91.408,5.020,24.652,-177.9923,31.7488,-4593.1434
C00578=-91.047,9.690,24.657,-177.0867,31.6111,-4596.0750
C00579=-90.755,13.981,24.767,179.6793,30.2766,-4598.7577
C00580=-91.008,16.781,25.041,172.1656,23.3532,-4600.4474
C00581=-91.772,18.686,25.406,171.5303,12.9811,-4601.5089
C00582=-92.865,20.265,25.771,174.8410,6.3558,-4602.3101
C00583=-94.037,21.871,26.043,177.5936,3.7116,-4603.0930
C00584=-94.948,23.861,26.175,179.2810,2.5691,-4604.1066
C00585=-95.323,26.720,26.245,179.9792,0.9711,-4605.6587
C00586=-95.074,30.093,26.301,179.9780,-0.1342,-4607.5637
C00587=-94.189,33.476,26.358,-179.9855,0.0427,-4609.5659
C00588=-93.020,36.693,26.395,-179.9984,0.0040,-4611.5274
C00589=-91.721,39.829,26.395,-179.9982,0.0040,-4613.4725
C00590=-90.273,42.931,26.358,-179.9801,0.0404,-4615.4343
C00591=-88.507,45.948,26.301,179.9207,-0.1105,-4617.4359
C00592=-86.297,48.509,26.245,-179.2986,0.6720,-4619.3411
C00593=-84.010,50.266,26.175,-177.6750,1.3092,-4620.8935
C00594=-81.959,51.029,26.043,-175.6775,0.9255,-4621.9071
C00595=-79.995,51.336,25.771,-171.8841,0.8549,-4622.6899
C00596=-78.105,51.679,25.406,-164.9814,3.3027,-4623.4910
C00597=-76.218,52.487,25.041,-158.0702,11.7507,-4624.5530
C00598=-74.059,54.287,24.767,-157.3747,22.2371,-4626.2423
C00599=-71.231,57.528,24.657,-158.2376,25.2298,-4628.9252
C00600=-68.184,61.085,24.652,-157.5713,24.8132,-4631.8567
C00601=-64.734,64.734,24.655,-156.3440,23.6556,-4635.0000
C00602=-61.085,68.184,24.652,-155.1871,22.4290,-4638.1433
C00603=-57.528,71.231,24.657,-154.7707,21.7628,-4641.0748
C00604=-54.287,74.059,24.767,-157.7626,22.6250,-4643.7577
C00605=-52.487,76.218,25.041,-168.2493,21.9298,-4645.4470
C00606=-51.679,78.105,25.406,-176.6973,15.0186,-4646.5090
C00607=-51.336,79.995,25.771,-179.1451,8.1159,-4647.3101
C00608=-51.029,81.959,26.043,-179.0745,4.3225,-4648.0929
C00609=-50.266,84.010,26.175,-178.6908,2.3250,-4649.1065
C00610=-48.509,86.297,26.245,-179.3280,0.7014,-4650.6589
C00611=-45.948,88.507,26.301,179.8895,-0.0793,-4652.5641
C00612=-42.931,90.273,26.358,-179.9596,0.0199,-4654.5657
C00613=-39.829,91.721,26.395,-179.9960,0.0018,-4656.5275
C00614=-36.693,93.020,26.395,-179.9960,0.0016,-4658.4726
C00615=-33.476,94.189,26.358,-179.9573,0.0145,-4660.4341
C00616=-30.093,95.074,26.301,179.8658,-0.0220,-4662.4363
C00617=-26.720,95.323,26.245,-179.0289,-0.0208,-4664.3413
C00618=-23.861,94.948,26.175,-177.4309,-0.7190,-4665.8934
C00619=-21.871,94.037,26.043,-176.2884,-2.4064,-4666.9070
C00620=-20.265,92.865,25.771,-173.6442,-5.1590,-4667.6899
C00621=-18.686,91.772,25.406,-167.0189,-8.4697,-4668.4911
C00622=-16.781,91.008,25.041,-156.6468,-7.8344,-4669.5526
C00623=-13.981,90.755,24.767,-149.7234,-0.3207,-4671.2423
C00624=-9.690,91.047,24.657,-148.3889,2.9133,-4673.9250
C00625=-5.020,91.408,24.652,-148.2512,2.0077,-4676.8566
C00626=0.000,91.548,24.655,-148.2220,0.0004,-4680.0000
C00627=0.000,90.369,26.513,-146.9909,0.0004,-4680.0000
C00628=4.912,90.233,26.509,-147.0206,-2.0967,-4683.1159
C00629=9.508,89.882,26.515,-147.1605,-2.8971,-4686.0385
C00630=13.759,89.629,26.645,-148.6809,1.2171,-4688.7274
C00631=16.509,89.983,26.968,-157.2655,9.5618,-4690.3963
C00632=18.373,90.901,27.402,-168.7365,8.8492,-4691.4267
C00633=19.923,92.196,27.838,-175.1312,4.7417,-4692.1938
C00634=21.502,93.597,28.166,-177.5251,1.9666,-4692.9380
C00635=23.458,94.728,28.327,-178.2716,0.6326,-4693.9087
C00636=26.340,95.277,28.411,-179.4215,0.0370,-4695.4538
C00637=29.791,95.129,28.479,179.6935,0.0440,-4697.3887
C00638=33.285,94.252,28.548,-179.9707,-0.0099,-4699.4506
C00639=36.628,93.045,28.594,-179.9976,-0.0009,-4701.4875
C00640=39.893,91.693,28.594,-179.9976,-0.0010,-4703.5125
C00641=43.110,90.182,28.548,-179.9723,-0.0138,-4705.5494
C00642=46.201,88.332,28.479,179.7522,0.1856,-4707.6113
C00643=48.746,85.996,28.411,-179.6171,-0.4352,-4709.5463
C00644=50.396,83.570,28.327,-179.2249,-1.6694,-4711.0916
C00645=50.979,81.387,28.166,-179.6401,-3.1392,-4712.0621
C00646=51.105,79.281,27.838,-179.9095,-6.7798,-4712.8061
C00647=51.285,77.269,27.402,-178.2394,-14.0854,-4713.5730
C00648=51.954,75.301,26.968,-169.9528,-22.5582,-4714.6038
C00649=53.649,73.106,26.645,-157.4504,-24.0022,-4716.2732
C00650=56.833,70.280,26.515,-153.7948,-22.8119,-4718.9613
C00651=60.331,67.277,26.509,-154.1393,-23.4102,-4721.8843
C00652=63.901,63.901,26.513,-155.3281,-24.6724,-4725.0000
C00653=67.277,60.331,26.509,-156.5894,-25.8604,-4728.1157
C00654=70.280,56.833,26.515,-157.1876,-26.2046,-4731.0387
C00655=73.106,53.649,26.645,-155.9981,-22.5500,-4733.7268
C00656=75.301,51.954,26.968,-157.4418,-10.0472,-4735.3962
C00657=77.269,51.285,27.402,-165.9146,-1.7606,-4736.4270
C00658=79.281,51.105,27.838,-173.2202,-0.0905,-4737.1939
C00659=81.387,50.979,28.166,-176.8608,-0.3599,-4737.9379
C00660=83.570,50.396,28.327,-178.3306,-0.7751,-4738.9084
C00661=85.996,48.746,28.411,-179.5648,-0.3829,-4740.4537
C00662=88.332,46.201,28.479,179.8144,0.2478,-4742.3887
C00663=90.182,43.110,28.548,-179.9862,-0.0277,-4744.4506
C00664=91.693,39.893,28.594,-179.9990,-0.0024,-4746.4875
C00665=93.045,36.628,28.594,-179.9991,-0.0024,-4748.5125
C00666=94.252,33.285,28.548,-179.9901,-0.0293,-4750.5494
C00667=95.129,29.791,28.479,179.9560,0.3065,-4752.6113
C00668=95.277,26.340,28.411,179.9630,-0.5785,-4754.5462
C00669=94.728,23.458,28.327,179.3674,-1.7284,-4756.0913
C00670=93.597,21.502,28.166,178.0334,-2.4749,-4757.0620
C00671=92.196,19.923,27.838,175.2583,-4.8688,-4757.8062
C00672=90.901,18.373,27.402,171.1508,-11.2635,-4758.5733
C00673=89.983,16.509,26.968,170.4382,-22.7345,-4759.6037
C00674=89.629,13.759,26.645,178.7829,-31.3191,-4761.2726
C00675=89.882,9.508,26.515,-177.1029,-32.8395,-4763.9615
C00676=90.233,4.912,26.509,-177.9033,-32.9794,-4766.8841
C00677=90.369,0.000,26.513,179.9996,-33.0091,-4770.0000
C00678=90.233,-4.912,26.509,177.9038,-32.9794,-4773.1159
C00679=89.882,-9.508,26.515,177.1039,-32.8395,-4776.0385
C00680=89.629,-13.759,26.645,-178.7835,-31.3192,-4778.7274
C00681=89.983,-16.509,26.968,-170.4382,-22.7345,-4780.3963
C00682=90.901,-18.373,27.402,-171.1508,-11.2635,-4781.4267
C00683=92.196,-19.923,27.838,-175.2583,-4.8688,-4782.1938
C00684=93.597,-21.502,28.166,-178.0334,-2.4749,-4782.9380
C00685=94.728,-23.458,28.327,-179.3674,-1.7284,-4783.9087
C00686=95.277,-26.340,28.411,-179.9630,-0.5785,-4785.4538
C00687=95.129,-29.791,28.479,-179.9560,0.3065,-4787.3887
C00688=94.252,-33.285,28.548,179.9901,-0.0293,-4789.4506
C00689=93.045,-36.628,28.594,179.9991,-0.0024,-4791.4875
C00690=91.693,-39.893,28.594,179.9990,-0.0024,-4793.5125
C00691=90.182,-43.110,28.548,179.9862,-0.0277,-4795.5494
C00692=88.332,-46.201,28.479,-179.8144,0.2478,-4797.6113
C00693=85.996,-48.746,28.411,179.5648,-0.3829,-4799.5463
C00694=83.570,-50.396,28.327,178.3306,-0.7751,-4801.0916
C00695=81.387,-50.979,28.166,176.8608,-0.3599,-4802.0621
C00696=79.281,-51.105,27.838,173.2202,-0.0905,-4802.8061
C00697=77.269,-51.285,27.402,165.9146,-1.7606,-4803.5730
C00698=75.301,-51.954,26.968,157.4418,-10.0472,-4804.6038
C00699=73.106,-53.649,26.645,155.9978,-22.5496,-4806.2732
C00700=70.280,-56.833,26.515,157.1881,-26.2052,-4808.9613
C00701=67.277,-60.331,26.509,156.5898,-25.8607,-4811.8843
C00702=63.901,-63.901,26.513,155.3276,-24.6719,-4815.0000
C00703=60.331,-67.277,26.509,154.1396,-23.4106,-4818.1157
C00704=56.833,-70.280,26.515,153.7954,-22.8124,-4821.0387
C00705=53.649,-73.106,26.645,157.4500,-24.0019,-4823.7268
C00706=51.954,-75.301,26.968,169.9528,-22.5582,-4825.3962
C00707=51.285,-77.269,27.402,178.2394,-14.0854,-4826.4270
C00708=51.105,-79.281,27.838,179.9095,-6.7798,-4827.1939
C00709=50.979,-81.387,28.166,179.6401,-3.1392,-4827.9379
C00710=50.396,-83.570,28.327,179.2249,-1.6694,-4828.9084
C00711=48.746,-85.996,28.411,179.6171,-0.4352,-4830.4537
C00712=46.201,-88.332,28.479,-179.7522,0.1856,-4832.3887
C00713=43.110,-90.182,28.548,179.9723,-0.0138,-4834.4506
C00714=39.893,-91.693,28.594,179.9976,-0.0010,-4836.4875
C00715=36.628,-93.045,28.594,179.9976,-0.0009,-4838.5125
C00716=33.285,-94.252,28.548,179.9707,-0.0099,-4840.5494
C00717=29.791,-95.129,28.479,-179.6935,0.0440,-4842.6113
C00718=26.340,-95.277,28.411,179.4215,0.0370,-4844.5462
C00719=23.458,-94.728,28.327,178.2716,0.6326,-4846.0913
C00720=21.502,-93.597,28.166,177.5251,1.9666,-4847.0620
C00721=19.923,-92.196,27.838,175.1312,4.7417,-4847.8062
C00722=18.373,-90.901,27.402,168.7365,8.8492,-4848.5733
C00723=16.509,-89.983,26.968,157.2655,9.5618,-4849.6037
C00724=13.759,-89.629,26.645,148.6809,1.2171,-4851.2726
C00725=9.508,-89.882,26.515,147.1605,-2.8971,-4853.9615
C00726=4.912,-90.233,26.509,147.0206,-2.0967,-4856.8841
C00727=0.000,-90.369,26.513,146.9909,0.0004,-4860.0000
C00728=0.000,-90.369,26.513,146.9909,0.0004,-4860.0000
C00729=-4.912,-90.233,26.509,147.0206,2.0962,-4863.1159
C00730=-9.508,-89.882,26.515,147.1605,2.8961,-4866.0385
C00731=-13.759,-89.629,26.645,148.6808,-1.2165,-4868.7274
C00732=-16.509,-89.983,26.968,157.2655,-9.5618,-4870.3963
C00733=-18.373,-90.901,27.402,168.7365,-8.8492,-4871.4267
C00734=-19.923,-92.196,27.838,175.1312,-4.7417,-4872.1938
C00735=-21.502,-93.597,28.166,177.5251,-1.9666,-4872.9380
C00736=-23.458,-94.728,28.327,178.2716,-0.6326,-4873.9087
C00737=-26.340,-95.277,28.411,179.4215,-0.0370,-4875.4538
C00738=-29.791,-95.129,28.479,-179.6935,-0.0440,-4877.3887
C00739=-33.285,-94.252,28.548,179.9707,0.0099,-4879.4506
C00740=-36.628,-93.045,28.594,179.9976,0.0009,-4881.4875
C00741=-39.893,-91.693,28.594,179.9976,0.0010,-4883.5125
C00742=-43.110,-90.182,28.548,179.9723,0.0138,-4885.5494
C00743=-46.201,-88.332,28.479,-179.7522,-0.1856,-4887.6113
C00744=-48.746,-85.996,28.411,179.6171,0.4352,-4889.5463
C00745=-50.396,-83.570,28.327,179.2249,1.6694,-4891.0916
C00746=-50.979,-81.387,28.166,179.6401,3.1392,-4892.0621
C00747=-51.105,-79.281,27.838,179.9095,6.7798,-4892.8061
C00748=-51.285,-77.269,27.402,178.2394,14.0854,-4893.5730
C00749=-51.954,-75.301,26.968,169.9528,22.5582,-4894.6038
C00750=-53.649,-73.106,26.645,157.4504,24.0022,-4896.2732
C00751=-56.833,-70.280,26.515,153.7948,22.8119,-4898.9613
C00752=-60.331,-67.277,26.509,154.1393,23.4102,-4901.8843
C00753=-63.901,-63.901,26.513,155.3281,24.6724,-4905.0000
C00754=-67.277,-60.331,26.509,156.5894,25.8604,-4908.1157
C00755=-70.280,-56.833,26.515,157.1876,26.2046,-4911.0387
C00756=-73.106,-53.649,26.645,155.9981,22.5500,-4913.7268
C00757=-75.301,-51.954,26.968,157.4418,10.0472,-4915.3962
C00758=-77.269,-51.285,27.402,165.9146,1.7606,-4916.4270
C00759=-79.281,-51.105,27.838,173.2202,0.0905,-4917.1939
C00760=-81.387,-50.979,28.166,176.8608,0.3599,-4917.9379
C00761=-83.570,-50.396,28.327,178.3306,0.7751,-4918.9084
C00762=-85.996,-48.746,28.411,179.5648,0.3829,-4920.4537
C00763=-88.332,-46.201,28.479,-179.8144,-0.2478,-4922.3887
C00764=-90.182,-43.110,28.548,179.9862,0.0277,-4924.4506
C00765=-91.693,-39.893,28.594,179.9990,0.0024,-4926.4875
C00766=-93.045,-36.628,28.594,179.9991,0.0024,-4928.5125
C00767=-94.252,-33.285,28.548,179.9901,0.0293,-4930.5494
C00768=-95.129,-29.791,28.479,-179.9560,-0.3065,-4932.6113
C00769=-95.277,-26.340,28.411,-179.9630,0.5785,-4934.5462
C00770=-94.728,-23.458,28.327,-179.3674,1.7284,-4936.0913
C00771=-93.597,-21.502,28.166,-178.0334,2.4749,-4937.0620
C00772=-92.196,-19.923,27.838,-175.2583,4.8688,-4937.8062
C00773=-90.901,-18.373,27.402,-171.1508,11.2635,-4938.5733
C00774=-89.983,-16.509,26.968,-170.4382,22.7345,-4939.6037
C00775=-89.629,-13.759,26.645,-178.7829,31.3191,-4941.2726
C00776=-89.882,-9.508,26.515,177.1029,32.8395,-4943.9615
C00777=-90.233,-4.912,26.509,177.9033,32.9794,-4946.8841
C00778=-90.369,0.000,26.513,-179.9996,33.0091,-4950.0000
C00779=-90.233,4.912,26.509,-177.9038,32.9794,-4953.1159
C00780=-89.882,9.508,26.515,-177.1039,32.8395,-4956.0385
C00781=-89.629,13.759,26.645,178.7835,31.3192,-4958.7274
C00782=-89.983,16.509,26.968,170.4382,22.7345,-4960.3963
C00783=-90.901,18.373,27.402,171.1508,11.2635,-4961.4267
C00784=-92.196,19.923,27.838,175.2583,4.8688,-4962.1938
C00785=-93.597,21.502,28.166,178.0334,2.4749,-4962.9380
C00786=-94.728,23.458,28.327,179.3674,1.7284,-4963.9087
C00787=-95.277,26.340,28.411,179.9630,0.5785,-4965.4538
C00788=-95.129,29.791,28.479,179.9560,-0.3065,-4967.3887
C00789=-94.252,33.285,28.548,-179.9901,0.0293,-4969.4506
C00790=-93.045,36.628,28.594,-179.9991,0.0024,-4971.4875
C00791=-91.693,39.893,28.594,-179.9990,0.0024,-4973.5125
C00792=-90.182,43.110,28.548,-179.9862,0.0277,-4975.5494
C00793=-88.332,46.201,28.479,179.8144,-0.2478,-4977.6113
C00794=-85.996,48.746,28.411,-179.5648,0.3829,-4979.5463
C00795=-83.570,50.396,28.327,-178.3306,0.7751,-4981.0916
C00796=-81.387,50.979,28.166,-176.8608,0.3599,-4982.0621
C00797=-79.281,51.105,27.838,-173.2202,0.0905,-4982.8061
C00798=-77.269,51.285,27.402,-165.9146,1.7606,-4983.5730
C00799=-75.301,51.954,26.968,-157.4418,10.0472,-4984.6038
C00800=-73.106,53.649,26.645,-155.9978,22.5496,-4986.2732
C00801=-70.280,56.833,26.515,-157.1881,26.2052,-4988.9613
C00802=-67.277,60.331,26.509,-156.5898,25.8607,-4991.8843
C00803=-63.901,63.901,26.513,-155.3276,24.6719,-4995.0000
C00804=-60.331,67.277,26.509,-154.1396,23.4106,-4998.1157
C00805=-56.833,70.280,26.515,-153.7954,22.8124,-5001.0387
C00806=-53.649,73.106,26.645,-157.4500,24.0019,-5003.7268
C00807=-51.954,75.301,26.968,-169.9528,22.5582,-5005.3962
C00808=-51.285,77.269,27.402,-178.2394,14.0854,-5006.4270
C00809=-51.105,79.281,27.838,-179.9095,6.7798,-5007.1939
C00810=-50.979,81.387,28.166,-179.6401,3.1392,-5007.9379
C00811=-50.396,83.570,28.327,-179.2249,1.6694,-5008.9084
C00812=-48.746,85.996,28.411,-179.6171,0.4352,-5010.4537
C00813=-46.201,88.332,28.479,179.7522,-0.1856,-5012.3887
C00814=-43.110,90.182,28.548,-179.9723,0.0138,-5014.4506
C00815=-39.893,91.693,28.594,-179.9976,0.0010,-5016.4875
C00816=-36.628,93.045,28.594,-179.9976,0.0009,-5018.5125
C00817=-33.285,94.252,28.548,-179.9707,0.0099,-5020.5494
C00818=-29.791,95.129,28.479,179.6935,-0.0440,-5022.6113
C00819=-26.340,95.277,28.411,-179.4215,-0.0370,-5024.5462
C00820=-23.458,94.728,28.327,-178.2716,-0.6326,-5026.0913
C00821=-21.502,93.597,28.166,-177.5251,-1.9666,-5027.0620
C00822=-19.923,92.196,27.838,-175.1312,-4.7417,-5027.8062
C00823=-18.373,90.901,27.402,-168.7365,-8.8492,-5028.5733
C00824=-16.509,89.983,26.968,-157.2655,-9.5618,-5029.6037
C00825=-13.759,89.629,26.645,-148.6808,-1.2165,-5031.2726
C00826=-9.508,89.882,26.515,-147.1605,2.8961,-5033.9615
C00827=-4.912,90.233,26.509,-147.0206,2.0962,-5036.8841
C00828=0.000,90.369,26.513,-146.9909,0.0004,-5040.0000
C00829=0.000,89.153,28.346,-145.9022,0.0004,-5040.0000
C00830=4.801,89.020,28.341,-145.9323,-2.1748,-5043.0871
C00831=9.321,88.681,28.348,-146.0749,-2.8439,-5046.0002
C00832=13.530,88.468,28.499,-147.8255,2.2168,-5048.6952
C00833=16.227,88.922,28.874,-158.3138,11.0586,-5050.3419
C00834=18.049,89.999,29.382,-170.5154,8.7916,-5051.3400
C00835=19.567,91.502,29.895,-176.4765,4.0373,-5052.0705
C00836=21.117,93.139,30.283,-178.6645,1.2702,-5052.7745
C00837=23.038,94.499,30.474,-179.1703,0.3790,-5053.7009
C00838=25.943,95.229,30.574,-179.8563,0.0154,-5055.2391
C00839=29.476,95.186,30.656,179.5089,0.0604,-5057.2060
C00840=33.085,94.318,30.738,-179.9851,-0.0050,-5059.3299
C00841=36.560,93.071,30.793,-179.9993,-0.0003,-5061.4458
C00842=39.959,91.663,30.793,-179.9994,-0.0003,-5063.5540
C00843=43.298,90.088,30.738,-179.9860,-0.0070,-5065.6698
C00844=46.464,88.150,30.656,179.6100,0.3045,-5067.7938
C00845=48.993,85.682,30.574,-179.9092,-0.1125,-5069.7609
C00846=50.531,83.111,30.474,-179.6813,-0.8547,-5071.2994
C00847=50.927,80.791,30.283,-179.9538,-1.8423,-5072.2255
C00848=50.865,78.538,29.895,179.6351,-5.3387,-5072.9290
C00849=50.876,76.401,29.382,-179.4973,-12.8163,-5073.6599
C00850=51.403,74.351,28.874,-171.8620,-22.7528,-5074.6583
C00851=52.989,72.123,28.499,-157.3406,-25.2777,-5076.3048
C00852=56.115,69.298,28.348,-152.9451,-23.7726,-5078.9993
C00853=59.552,66.342,28.341,-153.2053,-24.2903,-5081.9128
C00854=63.040,63.040,28.346,-154.4195,-25.5810,-5085.0000
C00855=66.342,59.552,28.341,-155.7093,-26.7944,-5088.0872
C00856=69.298,56.115,28.348,-156.2269,-27.0542,-5091.0007
C00857=72.123,52.989,28.499,-154.7226,-22.6600,-5093.6952
C00858=74.351,51.403,28.874,-157.2472,-8.1380,-5095.3417
C00859=76.401,50.876,29.382,-167.1837,-0.5027,-5096.3401
C00860=78.538,50.865,29.895,-174.6613,0.3649,-5097.0710
C00861=80.791,50.927,30.283,-178.1577,-0.0462,-5097.7745
C00862=83.111,50.531,30.474,-179.1453,-0.3187,-5098.7006
C00863=85.682,48.993,30.574,-179.8875,-0.0908,-5100.2391
C00864=88.150,46.464,30.656,179.6955,0.3900,-5102.2062
C00865=90.088,43.298,30.738,-179.9930,-0.0140,-5104.3302
C00866=91.663,39.959,30.793,-179.9997,-0.0006,-5106.4460
C00867=93.071,36.560,30.793,-179.9997,-0.0007,-5108.5542
C00868=94.318,33.085,30.738,-179.9950,-0.0149,-5110.6701
C00869=95.186,29.476,30.656,179.9396,0.4911,-5112.7940
C00870=95.229,25.943,30.574,179.9846,-0.1437,-5114.7609
C00871=94.499,23.038,30.474,179.6210,-0.8297,-5116.2991
C00872=93.139,21.117,30.283,178.7298,-1.3355,-5117.2255
C00873=91.502,19.567,29.895,175.9627,-3.5235,-5117.9295
C00874=89.999,18.049,29.382,171.2084,-9.4846,-5118.6600
C00875=88.922,16.227,28.874,168.9414,-21.6862,-5119.6581
C00876=88.468,13.530,28.499,177.7832,-32.1745,-5121.3048
C00877=88.681,9.321,28.348,-177.1561,-33.9251,-5123.9998
C00878=89.020,4.801,28.341,-177.8252,-34.0677,-5126.9129
C00879=89.153,0.000,28.346,179.9996,-34.0978,-5130.0000
C00880=89.020,-4.801,28.341,177.8258,-34.0678,-5133.0871
C00881=88.681,-9.321,28.348,177.1572,-33.9251,-5136.0002
C00882=88.468,-13.530,28.499,-177.7839,-32.1746,-5138.6952
C00883=88.922,-16.227,28.874,-168.9414,-21.6862,-5140.3419
C00884=89.999,-18.049,29.382,-171.2084,-9.4846,-5141.3400
C00885=91.502,-19.567,29.895,-175.9627,-3.5235,-5142.0705
C00886=93.139,-21.117,30.283,-178.7298,-1.3355,-5142.7745
C00887=94.499,-23.038,30.474,-179.6210,-0.8297,-5143.7009
C00888=95.229,-25.943,30.574,-179.9846,-0.1437,-5145.2391
C00889=95.186,-29.476,30.656,-179.9396,0.4911,-5147.2060
C00890=94.318,-33.085,30.738,179.9950,-0.0149,-5149.3299
C00891=93.071,-36.560,30.793,179.9997,-0.0007,-5151.4458
C00892=91.663,-39.959,30.793,179.9997,-0.0006,-5153.5540
C00893=90.088,-43.298,30.738,179.9930,-0.0140,-5155.6698
C00894=88.150,-46.464,30.656,-179.6955,0.3900,-5157.7938
C00895=85.682,-48.993,30.574,179.8875,-0.0908,-5159.7609
C00896=83.111,-50.531,30.474,179.1453,-0.3187,-5161.2994
C00897=80.791,-50.927,30.283,178.1577,-0.0462,-5162.2255
C00898=78.538,-50.865,29.895,174.6613,0.3649,-5162.9290
C00899=76.401,-50.876,29.382,167.1837,-0.5027,-5163.6599
C00900=74.351,-51.403,28.874,157.2472,-8.1380,-5164.6583
C00901=72.123,-52.989,28.499,154.7223,-22.6594,-5166.3048
C00902=69.298,-56.115,28.348,156.2274,-27.0549,-5168.9993
C00903=66.342,-59.552,28.341,155.7097,-26.7947,-5171.9128
C00904=63.040,-63.040,28.346,154.4190,-25.5805,-5175.0000
C00905=59.552,-66.342,28.341,153.2056,-24.2907,-5178.0872
C00906=56.115,-69.298,28.348,152.9458,-23.7731,-5181.0007
C00907=52.989,-72.123,28.499,157.3400,-25.2774,-5183.6952
C00908=51.403,-74.351,28.874,171.8620,-22.7528,-5185.3417
C00909=50.876,-76.401,29.382,179.4973,-12.8163,-5186.3401
C00910=50.865,-78.538,29.895,-179.6351,-5.3387,-5187.0710
C00911=50.927,-80.791,30.283,179.9538,-1.8423,-5187.7745
C00912=50.531,-83.111,30.474,179.6813,-0.8547,-5188.7006
C00913=48.993,-85.682,30.574,179.9092,-0.1125,-5190.2391
C00914=46.464,-88.150,30.656,-179.6100,0.3045,-5192.2062
C00915=43.298,-90.088,30.738,179.9860,-0.0070,-5194.3302
C00916=39.959,-91.663,30.793,179.9994,-0.0003,-5196.4460
C00917=36.560,-93.071,30.793,179.9993,-0.0003,-5198.5542
C00918=33.085,-94.318,30.738,179.9851,-0.0050,-5200.6701
C00919=29.476,-95.186,30.656,-179.5089,0.0604,-5202.7940
C00920=25.943,-95.229,30.574,179.8563,0.0154,-5204.7609
C00921=23.038,-94.499,30.474,179.1703,0.3790,-5206.2991
C00922=21.117,-93.139,30.283,178.6645,1.2702,-5207.2255
C00923=19.567,-91.502,29.895,176.4765,4.0373,-5207.9295
C00924=18.049,-89.999,29.382,170.5154,8.7916,-5208.6600
C00925=16.227,-88.922,28.874,158.3138,11.0586,-5209.6581
C00926=13.530,-88.468,28.499,147.8255,2.2168,-5211.3048
C00927=9.321,-88.681,28.348,146.0749,-2.8439,-5213.9998
C00928=4.801,-89.020,28.341,145.9323,-2.1748,-5216.9129
C00929=0.000,-89.153,28.346,145.9022,0.0004,-5220.0000
C00930=0.000,-89.153,28.346,145.9022,0.0004,-5220.0000
C00931=-4.801,-89.020,28.341,145.9322,2.1742,-5223.0871
C00932=-9.321,-88.681,28.348,146.0749,2.8428,-5226.0002
C00933=-13.530,-88.468,28.499,147.8254,-2.2161,-5228.6952
C00934=-16.227,-88.922,28.874,158.3138,-11.0586,-5230.3419
C00935=-18.049,-89.999,29.382,170.5154,-8.7916,-5231.3400
C00936=-19.567,-91.502,29.895,176.4765,-4.0373,-5232.0705
C00937=-21.117,-93.139,30.283,178.6645,-1.2702,-5232.7745
C00938=-23.038,-94.499,30.474,179.1703,-0.3790,-5233.7009
C00939=-25.943,-95.229,30.574,179.8563,-0.0154,-5235.2391
C00940=-29.476,-95.186,30.656,-179.5089,-0.0604,-5237.2060
C00941=-33.085,-94.318,30.738,179.9851,0.0050,-5239.3299
C00942=-36.560,-93.071,30.793,179.9993,0.0003,-5241.4458
C00943=-39.959,-91.663,30.793,179.9994,0.0003,-5243.5540
C00944=-43.298,-90.088,30.738,179.9860,0.0070,-5245.6698
C00945=-46.464,-88.150,30.656,-179.6100,-0.3045,-5247.7938
C00946=-48.993,-85.682,30.574,179.9092,0.1125,-5249.7609
C00947=-50.531,-83.111,30.474,179.6813,0.8547,-5251.2994
C00948=-50.927,-80.791,30.283,179.9538,1.8423,-5252.2255
C00949=-50.865,-78.538,29.895,-179.6351,5.3387,-5252.9290
C00950=-50.876,-76.401,29.382,179.4973,12.8163,-5253.6599
C00951=-51.403,-74.351,28.874,171.8620,22.7528,-5254.6583
C00952=-52.989,-72.123,28.499,157.3406,25.2777,-5256.3048
C00953=-56.115,-69.298,28.348,152.9451,23.7726,-5258.9993
C00954=-59.552,-66.342,28.341,153.2053,24.2903,-5261.9128
C00955=-63.040,-63.040,28.346,154.4195,25.5810,-5265.0000
C00956=-66.342,-59.552,28.341,155.7093,26.7944,-5268.0872
C00957=-69.298,-56.115,28.348,156.2269,27.0542,-5271.0007
C00958=-72.123,-52.989,28.499,154.7226,22.6600,-5273.6952
C00959=-74.351,-51.403,28.874,157.2472,8.1380,-5275.3417
C00960=-76.401,-50.876,29.382,167.1837,0.5027,-5276.3401
C00961=-78.538,-50.865,29.895,174.6613,-0.3649,-5277.0710
C00962=-80.791,-50.927,30.283,178.1577,0.0462,-5277.7745
C00963=-83.111,-50.531,30.474,179.1453,0.3187,-5278.7006
C00964=-85.682,-48.993,30.574,179.8875,0.0908,-5280.2391
C00965=-88.150,-46.464,30.656,-179.6955,-0.3900,-5282.2062
C00966=-90.088,-43.298,30.738,179.9930,0.0140,-5284.3302
C00967=-91.663,-39.959,30.793,179.9997,0.0006,-5286.4460
C00968=-93.071,-36.560,30.793,179.9997,0.0007,-5288.5542
C00969=-94.318,-33.085,30.738,179.9950,0.0149,-5290.6701
C00970=-95.186,-29.476,30.656,-179.9396,-0.4911,-5292.7940
C00971=-95.229,-25.943,30.574,-179.9846,0.1437,-5294.7609
C00972=-94.499,-23.038,30.474,-179.6210,0.8297,-5296.2991
C00973=-93.139,-21.117,30.283,-178.7298,1.3355,-5297.2255
C00974=-91.502,-19.567,29.895,-175.9627,3.5235,-5297.9295
C00975=-89.999,-18.049,29.382,-171.2084,9.4846,-5298.6600
C00976=-88.922,-16.227,28.874,-168.9414,21.6862,-5299.6581
C00977=-88.468,-13.530,28.499,-177.7832,32.1745,-5301.3048
C00978=-88.681,-9.321,28.348,177.1561,33.9251,-5303.9998
C00979=-89.020,-4.801,28.341,177.8252,34.0677,-5306.9129
C00980=-89.153,0.000,28.346,-179.9996,34.0978,-5310.0000
C00981=-89.020,4.801,28.341,-177.8258,34.0678,-5313.0871
C00982=-88.681,9.321,28.348,-177.1572,33.9251,-5316.0002
C00983=-88.468,13.530,28.499,177.7839,32.1746,-5318.6952
C00984=-88.922,16.227,28.874,168.9414,21.6862,-5320.3419
C00985=-89.999,18.049,29.382,171.2084,9.4846,-5321.3400
C00986=-91.502,19.567,29.895,175.9627,3.5235,-5322.0705
C00987=-93.139,21.117,30.283,178.7298,1.3355,-5322.7745
C00988=-94.499,23.038,30.474,179.6210,0.8297,-5323.7009
C00989=-95.229,25.943,30.574,179.9846,0.1437,-5325.2391
C00990=-95.186,29.476,30.656,179.9396,-0.4911,-5327.2060
C00991=-94.318,33.085,30.738,-179.9950,0.0149,-5329.3299
C00992=-93.071,36.560,30.793,-179.9997,0.0007,-5331.4458
C00993=-91.663,39.959,30.793,-179.9997,0.0006,-5333.5540
C00994=-90.088,43.298,30.738,-179.9930,0.0140,-5335.6698
C00995=-88.150,46.464,30.656,179.6955,-0.3900,-5337.7938
C00996=-85.682,48.993,30.574,-179.8875,0.0908,-5339.7609
C00997=-83.111,50.531,30.474,-179.1453,0.3187,-5341.2994
C00998=-80.791,50.927,30.283,-178.1577,0.0462,-5342.2255
C00999=-78.538,50.865,29.895,-174.6613,-0.3649,-5342.9290
C01000=-76.401,50.876,29.382,-167.1837,0.5027,-5343.6599
C01001=-74.351,51.403,28.874,-157.2472,8.1380,-5344.6583
C01002=-72.123,52.989,28.499,-154.7223,22.6594,-5346.3048
C01003=-69.298,56.115,28.348,-156.2274,27.0549,-5348.9993
C01004=-66.342,59.552,28.341,-155.7097,26.7947,-5351.9128
C01005=-63.040,63.040,28.346,-154.4190,25.5805,-5355.0000
C01006=-59.552,66.342,28.341,-153.2056,24.2907,-5358.0872
C01007=-56.115,69.298,28.348,-152.9458,23.7731,-5361.0007
C01008=-52.989,72.123,28.499,-157.3400,25.2774,-5363.6952
C01009=-51.403,74.351,28.874,-171.8620,22.7528,-5365.3417
C01010=-50.876,76.401,29.382,-179.4973,12.8163,-5366.3401
C01011=-50.865,78.538,29.895,179.6351,5.3387,-5367.0710
C01012=-50.927,80.791,30.283,-179.9538,1.8423,-5367.7745
C01013=-50.531,83.111,30.474,-179.6813,0.8547,-5368.7006
C01014=-48.993,85.682,30.574,-179.9092,0.1125,-5370.2391
C01015=-46.464,88.150,30.656,179.6100,-0.3045,-5372.2062
C01016=-43.298,90.088,30.738,-179.9860,0.0070,-5374.3302
C01017=-39.959,91.663,30.793,-179.9994,0.0003,-5376.4460
C01018=-36.560,93.071,30.793,-179.9993,0.0003,-5378.5542
C01019=-33.085,94.318,30.738,-179.9851,0.0050,-5380.6701
C01020=-29.476,95.186,30.656,179.5089,-0.0604,-5382.7940
C01021=-25.943,95.229,30.574,-179.8563,-0.0154,-5384.7609
C01022=-23.038,94.499,30.474,-179.1703,-0.3790,-5386.2991
C01023=-21.117,93.139,30.283,-178.6645,-1.2702,-5387.2255
C01024=-19.567,91.502,29.895,-176.4765,-4.0373,-5387.9295
C01025=-18.049,89.999,29.382,-170.5154,-8.7916,-5388.6600
C01026=-16.227,88.922,28.874,-158.3138,-11.0586,-5389.6581
C01027=-13.530,88.468,28.499,-147.8254,-2.2161,-5391.3048
C01028=-9.321,88.681,28.348,-146.0749,2.8428,-5393.9998
C01029=-4.801,89.020,28.341,-145.9322,2.1742,-5396.9129
C01030=0.000,89.153,28.346,-145.9022,0.0004,-5400.0000
C01031=0.000,87.904,30.157,-144.9432,0.0004,-5400.0000
C01032=4.687,87.776,30.152,-144.9734,-2.2427,-5403.0565
C01033=9.129,87.447,30.160,-145.1196,-2.7561,-5405.9598
C01034=13.294,87.274,30.332,-147.1504,3.3033,-5408.6610
C01035=15.938,87.830,30.762,-159.7282,12.2356,-5410.2852
C01036=17.714,89.068,31.347,-172.2272,8.3691,-5411.2483
C01037=19.200,90.783,31.942,-177.6276,3.1482,-5411.9417
C01038=20.718,92.664,32.394,-179.6431,0.3988,-5412.6030
C01039=22.602,94.262,32.617,179.9322,-0.0374,-5413.4837
C01040=25.531,95.180,32.735,179.6818,-0.0477,-5415.0155
C01041=29.149,95.246,32.831,179.3160,0.0705,-5417.0162
C01042=32.878,94.386,32.928,179.9997,0.0001,-5419.2050
C01043=36.490,93.098,32.991,179.9988,0.0004,-5421.4028
C01044=40.028,91.633,32.991,179.9989,0.0005,-5423.5971
C01045=43.493,89.989,32.928,179.9997,0.0001,-5425.7952
C01046=46.737,87.960,32.831,179.4665,0.4338,-5427.9837
C01047=49.249,85.356,32.735,179.8087,0.2587,-5429.9842
C01048=50.671,82.635,32.617,179.9785,0.0744,-5431.5162
C01049=50.874,80.174,32.394,179.9703,-0.5344,-5432.3970
C01050=50.617,77.770,31.942,179.4502,-3.9008,-5433.0583
C01051=50.455,75.506,31.347,179.5699,-11.3401,-5433.7518
C01052=50.836,73.375,30.762,-173.8456,-22.5147,-5434.7152
C01053=52.312,71.113,30.332,-157.4247,-26.4448,-5436.3389
C01054=55.379,68.290,30.160,-152.2123,-24.6497,-5439.0399
C01055=58.753,65.381,30.152,-152.3768,-25.0757,-5441.9437
C01056=62.157,62.157,30.157,-153.6112,-26.3893,-5445.0000
C01057=65.381,58.753,30.152,-154.9239,-27.6229,-5448.0563
C01058=68.290,55.379,30.160,-155.3497,-27.7869,-5450.9601
C01059=71.113,52.312,30.332,-153.5556,-22.5759,-5453.6611
C01060=73.375,50.836,30.762,-157.4853,-6.1544,-5455.2848
C01061=75.506,50.455,31.347,-168.6599,0.4301,-5456.2482
C01062=77.770,50.617,31.942,-176.0992,0.5498,-5456.9417
C01063=80.174,50.874,32.394,-179.4656,0.0297,-5457.6030
C01064=82.635,50.671,32.617,179.9256,0.0215,-5458.4838
C01065=85.356,49.249,32.735,179.7413,0.1913,-5460.0158
C01066=87.960,46.737,32.831,179.5662,0.5335,-5462.0163
C01067=89.989,43.493,32.928,179.9999,0.0003,-5464.2048
C01068=91.633,40.028,32.991,179.9995,0.0011,-5466.4029
C01069=93.098,36.490,32.991,179.9996,0.0012,-5468.5972
C01070=94.386,32.878,32.928,179.9999,0.0003,-5470.7950
C01071=95.246,29.149,32.831,179.9295,0.6840,-5472.9838
C01072=95.180,25.531,32.735,-179.9523,0.3182,-5474.9845
C01073=94.262,22.602,32.617,-179.9626,0.0678,-5476.5163
C01074=92.664,20.718,32.394,179.6012,-0.3569,-5477.3970
C01075=90.783,19.200,31.942,176.8518,-2.3724,-5478.0583
C01076=89.068,17.714,31.347,171.6309,-7.7728,-5478.7517
C01077=87.830,15.938,30.762,167.7644,-20.2718,-5479.7148
C01078=87.274,13.294,30.332,176.6967,-32.8496,-5481.3390
C01079=87.447,9.129,30.160,-177.2439,-34.8804,-5484.0402
C01080=87.776,4.687,30.152,-177.7573,-35.0266,-5486.9435
C01081=87.904,0.000,30.157,179.9996,-35.0568,-5490.0000
C01082=87.776,-4.687,30.152,177.7578,-35.0266,-5493.0565
C01083=87.447,-9.130,30.160,177.2451,-34.8803,-5495.9604
C01084=87.274,-13.294,30.332,-176.6975,-32.8497,-5498.6610
C01085=87.830,-15.938,30.762,-167.7644,-20.2718,-5500.2852
C01086=89.068,-17.714,31.347,-171.6309,-7.7728,-5501.2483
C01087=90.783,-19.200,31.942,-176.8518,-2.3724,-5501.9417
C01088=92.664,-20.718,32.394,-179.6012,-0.3569,-5502.6030
C01089=94.262,-22.602,32.617,179.9626,0.0678,-5503.4837
C01090=95.180,-25.531,32.735,179.9523,0.3182,-5505.0155
C01091=95.246,-29.149,32.831,-179.9295,0.6840,-5507.0162
C01092=94.386,-32.878,32.928,-179.9999,0.0003,-5509.2050
C01093=93.098,-36.490,32.991,-179.9996,0.0012,-5511.4028
C01094=91.633,-40.028,32.991,-179.9995,0.0011,-5513.5971
C01095=89.989,-43.493,32.928,-179.9999,0.0003,-5515.7952
C01096=87.960,-46.737,32.831,-179.5662,0.5335,-5517.9837
C01097=85.356,-49.249,32.735,-179.7413,0.1913,-5519.9842
C01098=82.635,-50.671,32.617,-179.9256,0.0215,-5521.5162
C01099=80.174,-50.874,32.394,179.4656,0.0297,-5522.3970
C01100=77.770,-50.617,31.942,176.0992,0.5498,-5523.0583
C01101=75.506,-50.455,31.347,168.6599,0.4301,-5523.7518
C01102=73.375,-50.836,30.762,157.4853,-6.1544,-5524.7152
C01103=71.113,-52.312,30.332,153.5552,-22.5753,-5526.3389
C01104=68.290,-55.379,30.160,155.3503,-27.7877,-5529.0399
C01105=65.381,-58.753,30.152,154.9243,-27.6232,-5531.9437
C01106=62.157,-62.157,30.157,153.6107,-26.3888,-5535.0000
C01107=58.753,-65.381,30.152,152.3771,-25.0761,-5538.0563
C01108=55.379,-68.290,30.160,152.2131,-24.6503,-5540.9601
C01109=52.312,-71.113,30.332,157.4241,-26.4444,-5543.6611
C01110=50.836,-73.375,30.762,173.8456,-22.5147,-5545.2848
C01111=50.455,-75.506,31.347,-179.5699,-11.3401,-5546.2482
C01112=50.617,-77.770,31.942,-179.4502,-3.9008,-5546.9417
C01113=50.874,-80.174,32.394,-179.9703,-0.5344,-5547.6030
C01114=50.671,-82.635,32.617,-179.9785,0.0744,-5548.4838
C01115=49.249,-85.356,32.735,-179.8087,0.2587,-5550.0158
C01116=46.737,-87.960,32.831,-179.4665,0.4338,-5552.0163
C01117=43.493,-89.989,32.928,-179.9997,0.0001,-5554.2048
C01118=40.028,-91.633,32.991,-179.9989,0.0005,-5556.4029
C01119=36.490,-93.098,32.991,-179.9988,0.0004,-5558.5972
C01120=32.878,-94.386,32.928,-179.9997,0.0001,-5560.7950
C01121=29.149,-95.246,32.831,-179.3160,0.0705,-5562.9838
C01122=25.531,-95.180,32.735,-179.6818,-0.0477,-5564.9845
C01123=22.602,-94.262,32.617,-179.9322,-0.0374,-5566.5163
C01124=20.718,-92.664,32.394,179.6431,0.3988,-5567.3970
C01125=19.200,-90.783,31.942,177.6276,3.1482,-5568.0583
C01126=17.714,-89.068,31.347,172.2272,8.3691,-5568.7517
C01127=15.938,-87.830,30.762,159.7282,12.2356,-5569.7148
C01128=13.294,-87.274,30.332,147.1504,3.3033,-5571.3390
C01129=9.129,-87.447,30.160,145.1196,-2.7561,-5574.0402
C01130=4.687,-87.776,30.152,144.9734,-2.2427,-5576.9435
C01131=0.000,-87.904,30.157,144.9432,0.0004,-5580.0000
C01132=0.000,-87.904,30.157,144.9432,0.0004,-5580.0000
C01133=-4.687,-87.776,30.152,144.9734,2.2422,-5583.0565
C01134=-9.130,-87.447,30.160,145.1197,2.7549,-5585.9604
C01135=-13.294,-87.274,30.332,147.1503,-3.3025,-5588.6610
C01136=-15.938,-87.830,30.762,159.7282,-12.2356,-5590.2852
C01137=-17.714,-89.068,31.347,172.2272,-8.3691,-5591.2483
C01138=-19.200,-90.783,31.942,177.6276,-3.1482,-5591.9417
C01139=-20.718,-92.664,32.394,179.6431,-0.3988,-5592.6030
C01140=-22.602,-94.262,32.617,-179.9322,0.0374,-5593.4837
C01141=-25.531,-95.180,32.735,-179.6818,0.0477,-5595.0155
C01142=-29.149,-95.246,32.831,-179.3160,-0.0705,-5597.0162
C01143=-32.878,-94.386,32.928,-179.9997,-0.0001,-5599.2050
C01144=-36.490,-93.098,32.991,-179.9988,-0.0004,-5601.4028
C01145=-40.028,-91.633,32.991,-179.9989,-0.0005,-5603.5971
C01146=-43.493,-89.989,32.928,-179.9997,-0.0001,-5605.7952
C01147=-46.737,-87.960,32.831,-179.4665,-0.4338,-5607.9837
C01148=-49.249,-85.356,32.735,-179.8087,-0.2587,-5609.9842
C01149=-50.671,-82.635,32.617,-179.9785,-0.0744,-5611.5162
C01150=-50.874,-80.174,32.394,-179.9703,0.5344,-5612.3970
C01151=-50.617,-77.770,31.942,-179.4502,3.9008,-5613.0583
C01152=-50.455,-75.506,31.347,-179.5699,11.3401,-5613.7518
C01153=-50.836,-73.375,30.762,173.8456,22.5147,-5614.7152
C01154=-52.312,-71.113,30.332,157.4247,26.4448,-5616.3389
C01155=-55.379,-68.290,30.160,152.2123,24.6497,-5619.0399
C01156=-58.753,-65.381,30.152,152.3768,25.0757,-5621.9437
C01157=-62.157,-62.157,30.157,153.6112,26.3893,-5625.0000
C01158=-65.381,-58.753,30.152,154.9239,27.6229,-5628.0563
C01159=-68.290,-55.379,30.160,155.3497,27.7869,-5630.9601
C01160=-71.113,-52.312,30.332,153.5556,22.5759,-5633.6611
C01161=-73.375,-50.836,30.762,157.4853,6.1544,-5635.2848
C01162=-75.506,-50.455,31.347,168.6599,-0.4301,-5636.2482
C01163=-77.770,-50.617,31.942,176.0992,-0.5498,-5636.9417
C01164=-80.174,-50.874,32.394,179.4656,-0.0297,-5637.6030
C01165=-82.635,-50.671,32.617,-179.9256,-0.0215,-5638.4838
C01166=-85.356,-49.249,32.735,-179.7413,-0.1913,-5640.0158
C01167=-87.960,-46.737,32.831,-179.5662,-0.5335,-5642.0163
C01168=-89.989,-43.493,32.928,-179.9999,-0.0003,-5644.2048
C01169=-91.633,-40.028,32.991,-179.9995,-0.0011,-5646.4029
C01170=-93.098,-36.490,32.991,-179.9996,-0.0012,-5648.5972
C01171=-94.386,-32.878,32.928,-179.9999,-0.0003,-5650.7950
C01172=-95.246,-29.149,32.831,-179.9295,-0.6840,-5652.9838
C01173=-95.180,-25.531,32.735,179.9523,-0.3182,-5654.9845
C01174=-94.262,-22.602,32.617,179.9626,-0.0678,-5656.5163
C01175=-92.664,-20.718,32.394,-179.6012,0.3569,-5657.3970
C01176=-90.783,-19.200,31.942,-176.8518,2.3724,-5658.0583
C01177=-89.068,-17.714,31.347,-171.6309,7.7728,-5658.7517
C01178=-87.830,-15.938,30.762,-167.7644,20.2718,-5659.7148
C01179=-87.274,-13.294,30.332,-176.6967,32.8496,-5661.3390
C01180=-87.447,-9.129,30.160,177.2439,34.8804,-5664.0402
C01181=-87.776,-4.687,30.152,177.7573,35.0266,-5666.9435
C01182=-87.904,0.000,30.157,-179.9996,35.0568,-5670.0000
C01183=-87.776,4.687,30.152,-177.7578,35.0266,-5673.0565
C01184=-87.447,9.130,30.160,-177.2451,34.8803,-5675.9604
C01185=-87.274,13.294,30.332,176.6975,32.8497,-5678.6610
C01186=-87.830,15.938,30.762,167.7644,20.2718,-5680.2852
C01187=-89.068,17.714,31.347,171.6309,7.7728,-5681.2483
C01188=-90.783,19.200,31.942,176.8518,2.3724,-5681.9417
C01189=-92.664,20.718,32.394,179.6012,0.3569,-5682.6030
C01190=-94.262,22.602,32.617,-179.9626,-0.0678,-5683.4837
C01191=-95.180,25.531,32.735,-179.9523,-0.3182,-5685.0155
C01192=-95.246,29.149,32.831,179.9295,-0.6840,-5687.0162
C01193=-94.386,32.878,32.928,179.9999,-0.0003,-5689.2050
C01194=-93.098,36.490,32.991,179.9996,-0.0012,-5691.4028
C01195=-91.633,40.028,32.991,179.9995,-0.0011,-5693.5971
C01196=-89.989,43.493,32.928,179.9999,-0.0003,-5695.7952
C01197=-87.960,46.737,32.831,179.5662,-0.5335,-5697.9837
C01198=-85.356,49.249,32.735,179.7413,-0.1913,-5699.9842
C01199=-82.635,50.671,32.617,179.9256,-0.0215,-5701.5162
C01200=-80.174,50.874,32.394,-179.4656,-0.0297,-5702.3970
C01201=-77.770,50.617,31.942,-176.0992,-0.5498,-5703.0583
C01202=-75.506,50.455,31.347,-168.6599,-0.4301,-5703.7518
C01203=-73.375,50.836,30.762,-157.4853,6.1544,-5704.7152
C01204=-71.113,52.312,30.332,-153.5552,22.5753,-5706.3389
C01205=-68.290,55.379,30.160,-155.3503,27.7877,-5709.0399
C01206=-65.381,58.753,30.152,-154.9243,27.6232,-5711.9437
C01207=-62.157,62.157,30.157,-153.6107,26.3888,-5715.0000
C01208=-58.753,65.381,30.152,-152.3771,25.0761,-5718.0563
C01209=-55.379,68.290,30.160,-152.2131,24.6503,-5720.9601
C01210=-52.312,71.113,30.332,-157.4241,26.4444,-5723.6611
C01211=-50.836,73.375,30.762,-173.8456,22.5147,-5725.2848
C01212=-50.455,75.506,31.347,179.5699,11.3401,-5726.2482
C01213=-50.617,77.770,31.942,179.4502,3.9008,-5726.9417
C01214=-50.874,80.174,32.394,179.9703,0.5344,-5727.6030
C01215=-50.671,82.635,32.617,179.9785,-0.0744,-5728.4838
C01216=-49.249,85.356,32.735,179.8087,-0.2587,-5730.0158
C01217=-46.737,87.960,32.831,179.4665,-0.4338,-5732.0163
C01218=-43.493,89.989,32.928,179.9997,-0.0001,-5734.2048
C01219=-40.028,91.633,32.991,179.9989,-0.0005,-5736.4029
C01220=-36.490,93.098,32.991,179.9988,-0.0004,-5738.5972
C01221=-32.878,94.386,32.928,179.9997,-0.0001,-5740.7950
C01222=-29.149,95.246,32.831,179.3160,-0.0705,-5742.9838
C01223=-25.531,95.180,32.735,179.6818,0.0477,-5744.9845
C01224=-22.602,94.262,32.617,179.9322,0.0374,-5746.5163
C01225=-20.718,92.664,32.394,-179.6431,-0.3988,-5747.3970
C01226=-19.200,90.783,31.942,-177.6276,-3.1482,-5748.0583
C01227=-17.714,89.068,31.347,-172.2272,-8.3691,-5748.7517
C01228=-15.938,87.830,30.762,-159.7282,-12.2356,-5749.7148
C01229=-13.294,87.274,30.332,-147.1503,-3.3025,-5751.3390
C01230=-9.130,87.447,30.160,-145.1197,2.7549,-5754.0396
C01231=-4.687,87.776,30.152,-144.9734,2.2422,-5756.9435
C01232=0.000,87.904,30.157,-144.9432,0.0004,-5760.0000
C01233=0.000,86.627,31.948,-144.1028,0.0004,-5760.0000
C01234=4.570,86.503,31.943,-144.1331,-2.3009,-5763.0242
C01235=8.933,86.186,31.951,-144.2840,-2.6354,-5765.9175
C01236=13.053,86.053,32.146,-146.6498,4.4571,-5768.6252
C01237=15.641,86.712,32.633,-161.4230,13.0408,-5770.2250
C01238=17.370,88.113,33.299,-173.7884,7.6720,-5771.1519
C01239=18.822,90.045,33.980,-178.5738,2.1633,-5771.8065
C01240=20.308,92.176,34.500,179.5624,-0.5662,-5772.4248
C01241=22.152,94.017,34.757,179.0872,-0.5942,-5773.2580
C01242=25.107,95.129,34.893,179.2076,-0.1524,-5774.7847
C01243=28.812,95.307,35.004,179.1192,0.0737,-5776.8204
C01244=32.664,94.457,35.116,179.9841,0.0052,-5779.0758
C01245=36.417,93.126,35.190,179.9970,0.0012,-5781.3580
C01246=40.099,91.601,35.190,179.9971,0.0013,-5783.6417
C01247=43.694,89.888,35.116,179.9851,0.0076,-5785.9241
C01248=47.019,87.765,35.004,179.3251,0.5708,-5788.1796
C01249=49.513,85.019,34.893,179.5474,0.6681,-5790.2155
C01250=50.816,82.144,34.757,179.7747,1.0655,-5791.7418
C01251=50.818,79.538,34.500,-179.9091,0.7097,-5792.5751
C01252=50.362,76.980,33.980,179.4783,-2.5374,-5793.1936
C01253=50.022,74.588,33.299,178.9521,-9.7713,-5793.8475
C01254=50.255,72.374,32.633,-175.7750,-21.8720,-5794.7753
C01255=51.619,70.079,32.146,-157.6940,-27.4964,-5796.3747
C01256=54.626,67.259,31.951,-151.5886,-25.4479,-5799.0826
C01257=57.935,64.399,31.943,-151.6465,-25.7724,-5801.9754
C01258=61.254,61.254,31.948,-152.8966,-27.1039,-5805.0000
C01259=64.398,57.936,31.943,-154.2272,-28.3532,-5808.0237
C01260=67.259,54.626,31.951,-154.5515,-28.4105,-5810.9174
C01261=70.079,51.619,32.146,-152.5039,-22.3066,-5813.6253
C01262=72.374,50.255,32.633,-158.1280,-4.2250,-5815.2247
C01263=74.588,50.022,33.299,-170.2287,1.0479,-5816.1525
C01264=76.980,50.362,33.980,-177.4626,0.5217,-5816.8064
C01265=79.538,50.818,34.500,179.2903,-0.0909,-5817.4249
C01266=82.144,50.816,34.757,178.9345,0.2253,-5818.2582
C01267=85.019,49.513,34.893,179.3319,0.4526,-5819.7845
C01268=87.765,47.019,35.004,179.4292,0.6749,-5821.8204
C01269=89.888,43.694,35.116,179.9924,0.0149,-5824.0759
C01270=91.601,40.099,35.190,179.9987,0.0029,-5826.3583
C01271=93.126,36.417,35.190,179.9988,0.0030,-5828.6420
C01272=94.457,32.664,35.116,179.9948,0.0159,-5830.9242
C01273=95.307,28.812,35.004,179.9263,0.8808,-5833.1796
C01274=95.129,25.107,34.893,-179.8476,0.7924,-5835.2153
C01275=94.017,22.152,34.757,-179.4058,0.9128,-5836.7420
C01276=92.176,20.308,34.500,-179.4338,0.4376,-5837.5752
C01277=90.045,18.822,33.980,177.8367,-1.4262,-5838.1935
C01278=88.113,17.370,33.299,172.3280,-6.2116,-5838.8481
C01279=86.712,15.641,32.633,166.9592,-18.5770,-5839.7750
C01280=86.053,13.053,32.146,175.5429,-33.3502,-5841.3748
C01281=86.186,8.933,31.951,-177.3646,-35.7160,-5844.0825
C01282=86.503,4.570,31.943,-177.6991,-35.8669,-5846.9758
C01283=86.627,0.000,31.948,179.9996,-35.8972,-5850.0000
C01284=86.503,-4.570,31.943,177.6997,-35.8669,-5853.0242
C01285=86.186,-8.933,31.951,177.3659,-35.7159,-5855.9175
C01286=86.053,-13.053,32.146,-175.5437,-33.3504,-5858.6252
C01287=86.712,-15.641,32.633,-166.9592,-18.5770,-5860.2250
C01288=88.113,-17.370,33.299,-172.3280,-6.2116,-5861.1519
C01289=90.045,-18.822,33.980,-177.8367,-1.4262,-5861.8065
C01290=92.176,-20.308,34.500,179.4338,0.4376,-5862.4248
C01291=94.017,-22.152,34.757,179.4058,0.9128,-5863.2580
C01292=95.129,-25.107,34.893,179.8476,0.7924,-5864.7847
C01293=95.307,-28.812,35.004,-179.9263,0.8808,-5866.8204
C01294=94.457,-32.664,35.116,-179.9948,0.0159,-5869.0758
C01295=93.126,-36.417,35.190,-179.9988,0.0030,-5871.3580
C01296=91.601,-40.099,35.190,-179.9987,0.0029,-5873.6417
C01297=89.888,-43.694,35.116,-179.9924,0.0149,-5875.9241
C01298=87.765,-47.019,35.004,-179.4292,0.6749,-5878.1796
C01299=85.019,-49.513,34.893,-179.3319,0.4526,-5880.2155
C01300=82.144,-50.816,34.757,-178.9345,0.2253,-5881.7418
C01301=79.538,-50.818,34.500,-179.2903,-0.0909,-5882.5751
C01302=76.980,-50.362,33.980,177.4626,0.5217,-5883.1936
C01303=74.588,-50.022,33.299,170.2287,1.0479,-5883.8475
C01304=72.374,-50.255,32.633,158.1280,-4.2250,-5884.7753
C01305=70.079,-51.619,32.146,152.5036,-22.3060,-5886.3747
C01306=67.259,-54.626,31.951,154.5521,-28.4114,-5889.0826
C01307=64.399,-57.935,31.943,154.2276,-28.3535,-5891.9754
C01308=61.254,-61.254,31.948,152.8961,-27.1034,-5895.0000
C01309=57.936,-64.398,31.943,151.6468,-25.7728,-5898.0237
C01310=54.626,-67.259,31.951,151.5895,-25.4485,-5900.9174
C01311=51.619,-70.079,32.146,157.6934,-27.4961,-5903.6253
C01312=50.255,-72.374,32.633,175.7750,-21.8720,-5905.2247
C01313=50.022,-74.588,33.299,-178.9521,-9.7713,-5906.1525
C01314=50.362,-76.980,33.980,-179.4783,-2.5374,-5906.8064
C01315=50.818,-79.538,34.500,179.9091,0.7097,-5907.4249
C01316=50.816,-82.144,34.757,-179.7747,1.0655,-5908.2582
C01317=49.513,-85.019,34.893,-179.5474,0.6681,-5909.7845
C01318=47.019,-87.765,35.004,-179.3251,0.5708,-5911.8204
C01319=43.694,-89.888,35.116,-179.9851,0.0076,-5914.0759
C01320=40.099,-91.601,35.190,-179.9971,0.0013,-5916.3583
C01321=36.417,-93.126,35.190,-179.9970,0.0012,-5918.6420
C01322=32.664,-94.457,35.116,-179.9841,0.0052,-5920.9242
C01323=28.812,-95.307,35.004,-179.1192,0.0737,-5923.1796
C01324=25.107,-95.129,34.893,-179.2076,-0.1524,-5925.2153
C01325=22.152,-94.017,34.757,-179.0872,-0.5942,-5926.7420
C01326=20.308,-92.176,34.500,-179.5624,-0.5662,-5927.5752
C01327=18.822,-90.045,33.980,178.5738,2.1633,-5928.1935
C01328=17.370,-88.113,33.299,173.7884,7.6720,-5928.8481
C01329=15.641,-86.712,32.633,161.4230,13.0408,-5929.7750
C01330=13.053,-86.053,32.146,146.6498,4.4571,-5931.3748
C01331=8.933,-86.186,31.951,144.2840,-2.6354,-5934.0825
C01332=4.570,-86.503,31.943,144.1331,-2.3009,-5936.9758
C01333=0.000,-86.627,31.948,144.1028,0.0004,-5940.0000
C01334=0.000,-86.627,31.948,144.1028,0.0004,-5940.0000
C01335=-4.570,-86.503,31.943,144.1331,2.3003,-5943.0242
C01336=-8.933,-86.186,31.951,144.2841,2.6341,-5945.9175
C01337=-13.053,-86.053,32.146,146.6496,-4.4563,-5948.6252
C01338=-15.641,-86.712,32.633,161.4230,-13.0408,-5950.2250
C01339=-17.370,-88.113,33.299,173.7884,-7.6720,-5951.1519
C01340=-18.822,-90.045,33.980,178.5738,-2.1633,-5951.8065
C01341=-20.308,-92.176,34.500,-179.5624,0.5662,-5952.4248
C01342=-22.152,-94.017,34.757,-179.0872,0.5942,-5953.2580
C01343=-25.107,-95.129,34.893,-179.2076,0.1524,-5954.7847
C01344=-28.812,-95.307,35.004,-179.1192,-0.0737,-5956.8204
C01345=-32.664,-94.457,35.116,-179.9841,-0.0052,-5959.0758
C01346=-36.417,-93.126,35.190,-179.9970,-0.0012,-5961.3580
C01347=-40.099,-91.601,35.190,-179.9971,-0.0013,-5963.6417
C01348=-43.694,-89.888,35.116,-179.9851,-0.0076,-5965.9241
C01349=-47.019,-87.765,35.004,-179.3251,-0.5708,-5968.1796
C01350=-49.513,-85.019,34.893,-179.5474,-0.6681,-5970.2155
C01351=-50.816,-82.144,34.757,-179.7747,-1.0655,-5971.7418
C01352=-50.818,-79.538,34.500,179.9091,-0.7097,-5972.5751
C01353=-50.362,-76.980,33.980,-179.4783,2.5374,-5973.1936
C01354=-50.022,-74.588,33.299,-178.9521,9.7713,-5973.8475
C01355=-50.255,-72.374,32.633,175.7750,21.8720,-5974.7753
C01356=-51.619,-70.079,32.146,157.6940,27.4964,-5976.3747
C01357=-54.626,-67.259,31.951,151.5886,25.4479,-5979.0826
C01358=-57.935,-64.399,31.943,151.6465,25.7724,-5981.9754
C01359=-61.254,-61.254,31.948,152.8966,27.1039,-5985.0000
C01360=-64.398,-57.936,31.943,154.2272,28.3532,-5988.0237
C01361=-67.259,-54.626,31.951,154.5515,28.4105,-5990.9174
C01362=-70.079,-51.619,32.146,152.5039,22.3066,-5993.6253
C01363=-72.374,-50.255,32.633,158.1280,4.2250,-5995.2247
C01364=-74.588,-50.022,33.299,170.2287,-1.0479,-5996.1525
C01365=-76.980,-50.362,33.980,177.4626,-0.5217,-5996.8064
C01366=-79.538,-50.818,34.500,-179.2903,0.0909,-5997.4249
C01367=-82.144,-50.816,34.757,-178.9345,-0.2253,-5998.2582
C01368=-85.019,-49.513,34.893,-179.3319,-0.4526,-5999.7845
C01369=-87.765,-47.019,35.004,-179.4292,-0.6749,-6001.8204
C01370=-89.888,-43.694,35.116,-179.9924,-0.0149,-6004.0759
C01371=-91.601,-40.099,35.190,-179.9987,-0.0029,-6006.3583
C01372=-93.126,-36.417,35.190,-179.9988,-0.0030,-6008.6420
C01373=-94.457,-32.664,35.116,-179.9948,-0.0159,-6010.9242
C01374=-95.307,-28.812,35.004,-179.9263,-0.8808,-6013.1796
C01375=-95.129,-25.107,34.893,179.8476,-0.7924,-6015.2153
C01376=-94.017,-22.152,34.757,179.4058,-0.9128,-6016.7420
C01377=-92.176,-20.308,34.500,179.4338,-0.4376,-6017.5752
C01378=-90.045,-18.822,33.980,-177.8367,1.4262,-6018.1935
C01379=-88.113,-17.370,33.299,-172.3280,6.2116,-6018.8481
C01380=-86.712,-15.641,32.633,-166.9592,18.5770,-6019.7750
C01381=-86.053,-13.053,32.146,-175.5429,33.3502,-6021.3748
C01382=-86.186,-8.933,31.951,177.3646,35.7160,-6024.0825
C01383=-86.503,-4.570,31.943,177.6991,35.8669,-6026.9758
C01384=-86.627,0.000,31.948,-179.9996,35.8972,-6030.0000
C01385=-86.503,4.570,31.943,-177.6997,35.8669,-6033.0242
C01386=-86.186,8.933,31.951,-177.3659,35.7159,-6035.9175
C01387=-86.053,13.053,32.146,175.5437,33.3504,-6038.6252
C01388=-86.712,15.641,32.633,166.9592,18.5770,-6040.2250
C01389=-88.113,17.370,33.299,172.3280,6.2116,-6041.1519
C01390=-90.045,18.822,33.980,177.8367,1.4262,-6041.8065
C01391=-92.176,20.308,34.500,-179.4338,-0.4376,-6042.4248
C01392=-94.017,22.152,34.757,-179.4058,-0.9128,-6043.2580
C01393=-95.129,25.107,34.893,-179.8476,-0.7924,-6044.7847
C01394=-95.307,28.812,35.004,179.9263,-0.8808,-6046.8204
C01395=-94.457,32.664,35.116,179.9948,-0.0159,-6049.0758
C01396=-93.126,36.417,35.190,179.9988,-0.0030,-6051.3580
C01397=-91.601,40.099,35.190,179.9987,-0.0029,-6053.6417
C01398=-89.888,43.694,35.116,179.9924,-0.0149,-6055.9241
C01399=-87.765,47.019,35.004,179.4292,-0.6749,-6058.1796
C01400=-85.019,49.513,34.893,179.3319,-0.4526,-6060.2155
C01401=-82.144,50.816,34.757,178.9345,-0.2253,-6061.7418
C01402=-79.538,50.818,34.500,179.2903,0.0909,-6062.5751
C01403=-76.980,50.362,33.980,-177.4626,-0.5217,-6063.1936
C01404=-74.588,50.022,33.299,-170.2287,-1.0479,-6063.8475
C01405=-72.374,50.255,32.633,-158.1280,4.2250,-6064.7753
C01406=-70.079,51.619,32.146,-152.5036,22.3060,-6066.3747
C01407=-67.259,54.626,31.951,-154.5521,28.4114,-6069.0826
C01408=-64.399,57.935,31.943,-154.2276,28.3535,-6071.9754
C01409=-61.254,61.254,31.948,-152.8961,27.1034,-6075.0000
C01410=-57.936,64.398,31.943,-151.6468,25.7728,-6078.0237
C01411=-54.626,67.259,31.951,-151.5895,25.4485,-6080.9174
C01412=-51.619,70.079,32.146,-157.6934,27.4961,-6083.6253
C01413=-50.255,72.374,32.633,-175.7750,21.8720,-6085.2247
C01414=-50.022,74.588,33.299,178.9521,9.7713,-6086.1525
C01415=-50.362,76.980,33.980,179.4783,2.5374,-6086.8064
C01416=-50.818,79.538,34.500,-179.9091,-0.7097,-6087.4249
C01417=-50.816,82.144,34.757,179.7747,-1.0655,-6088.2582
C01418=-49.513,85.019,34.893,179.5474,-0.6681,-6089.7845
C01419=-47.019,87.765,35.004,179.3251,-0.5708,-6091.8204
C01420=-43.694,89.888,35.116,179.9851,-0.0076,-6094.0759
C01421=-40.099,91.601,35.190,179.9971,-0.0013,-6096.3583
C01422=-36.417,93.126,35.190,179.9970,-0.0012,-6098.6420
C01423=-32.664,94.457,35.116,179.9841,-0.0052,-6100.9242
C01424=-28.812,95.307,35.004,179.1192,-0.0737,-6103.1796
C01425=-25.107,95.129,34.893,179.2076,0.1524,-6105.2153
C01426=-22.152,94.017,34.757,179.0872,0.5942,-6106.7420
C01427=-20.308,92.176,34.500,179.5624,0.5662,-6107.5752
C01428=-18.822,90.045,33.980,-178.5738,-2.1633,-6108.1935
C01429=-17.370,88.113,33.299,-173.7884,-7.6720,-6108.8481
C01430=-15.641,86.712,32.633,-161.4230,-13.0408,-6109.7750
C01431=-13.053,86.053,32.146,-146.6496,-4.4563,-6111.3748
C01432=-8.933,86.186,31.951,-144.2841,2.6341,-6114.0825
C01433=-4.570,86.503,31.943,-144.1331,2.3003,-6116.9758
C01434=0.000,86.627,31.948,-144.1028,0.0004,-6120.0000
C01435=0.000,85.325,33.722,-143.3716,0.0004,-6120.0000
C01436=4.451,85.206,33.716,-143.4019,-2.3496,-6122.9903
C01437=8.733,84.900,33.725,-143.5590,-2.4835,-6125.8729
C01438=12.808,84.808,33.943,-146.3185,5.6572,-6128.5881
C01439=15.338,85.570,34.490,-163.2997,13.4594,-6130.1621
C01440=17.019,87.137,35.239,-175.1574,6.7892,-6131.0515
C01441=18.435,89.289,36.009,-179.3291,1.1505,-6131.6656
C01442=19.887,91.675,36.600,178.9476,-1.5568,-6132.2395
C01443=21.692,93.766,36.894,178.3326,-1.2566,-6133.0258
C01444=24.671,95.076,37.049,178.7354,-0.2964,-6134.5467
C01445=28.465,95.370,37.176,178.9222,0.0699,-6136.6187
C01446=32.445,94.529,37.304,179.9684,0.0102,-6138.9437
C01447=36.342,93.155,37.389,179.9952,0.0018,-6141.3119
C01448=40.172,91.569,37.389,179.9953,0.0021,-6143.6874
C01449=43.901,89.784,37.304,179.9704,0.0151,-6146.0569
C01450=47.309,87.565,37.176,179.1885,0.7127,-6148.3812
C01451=49.784,84.674,37.049,179.3153,1.1038,-6150.4534
C01452=50.965,81.641,36.894,179.7094,2.0671,-6151.9748
C01453=50.762,78.886,36.600,-179.6431,1.8447,-6152.7607
C01454=50.101,76.172,36.009,179.6608,-1.2879,-6153.3343
C01455=49.580,73.649,35.239,178.6093,-8.1993,-6153.9482
C01456=49.662,71.353,34.490,-177.5427,-20.8758,-6154.8381
C01457=50.912,69.025,33.943,-158.1390,-28.4266,-6156.4120
C01458=53.858,66.209,33.725,-151.0673,-26.1712,-6159.1268
C01459=57.102,63.397,33.716,-151.0082,-26.3858,-6162.0095
C01460=60.334,60.334,33.722,-152.2699,-27.7306,-6165.0000
C01461=63.397,57.102,33.716,-153.6139,-28.9915,-6167.9905
C01462=66.209,53.858,33.725,-153.8281,-28.9318,-6170.8732
C01463=69.025,50.912,33.943,-151.5737,-21.8617,-6173.5880
C01464=71.353,49.662,34.490,-159.1242,-2.4573,-6175.1619
C01465=73.649,49.580,35.239,-171.8007,1.3907,-6176.0518
C01466=76.172,50.101,36.009,-178.7121,0.3392,-6176.6657
C01467=78.886,50.762,36.600,178.1553,-0.3569,-6177.2393
C01468=81.641,50.965,36.894,177.9329,0.2906,-6178.0252
C01469=84.674,49.784,37.049,178.8962,0.6847,-6179.5466
C01470=87.565,47.309,37.176,179.2873,0.8115,-6181.6188
C01471=89.784,43.901,37.304,179.9849,0.0296,-6183.9431
C01472=91.569,40.172,37.389,179.9979,0.0047,-6186.3126
C01473=93.155,36.342,37.389,179.9982,0.0048,-6188.6881
C01474=94.529,32.445,37.304,179.9898,0.0316,-6191.0563
C01475=95.370,28.465,37.176,179.9301,1.0778,-6193.3813
C01476=95.076,24.671,37.049,-179.7036,1.2646,-6195.4533
C01477=93.766,21.692,36.894,-178.7434,1.6674,-6196.9742
C01478=91.675,19.887,36.600,-178.4432,1.0524,-6197.7605
C01479=89.289,18.435,36.009,178.8495,-0.6709,-6198.3344
C01480=87.137,17.019,35.239,173.2108,-4.8426,-6198.9485
C01481=85.570,15.338,34.490,166.5406,-16.7003,-6199.8379
C01482=84.808,12.808,33.943,174.3428,-33.6815,-6201.4119
C01483=84.900,8.733,33.725,-177.5165,-36.4410,-6204.1271
C01484=85.206,4.451,33.716,-177.6504,-36.5981,-6207.0097
C01485=85.325,0.000,33.722,179.9996,-36.6284,-6210.0000
C01486=85.206,-4.451,33.716,177.6510,-36.5982,-6212.9903
C01487=84.900,-8.733,33.725,177.5180,-36.4409,-6215.8729
C01488=84.808,-12.808,33.943,-174.3436,-33.6818,-6218.5881
C01489=85.570,-15.338,34.490,-166.5406,-16.7003,-6220.1621
C01490=87.137,-17.019,35.239,-173.2108,-4.8426,-6221.0515
C01491=89.289,-18.435,36.009,-178.8495,-0.6709,-6221.6656
C01492=91.675,-19.887,36.600,178.4432,1.0524,-6222.2395
C01493=93.766,-21.692,36.894,178.7434,1.6674,-6223.0258
C01494=95.076,-24.671,37.049,179.7036,1.2646,-6224.5467
C01495=95.370,-28.465,37.176,-179.9301,1.0778,-6226.6187
C01496=94.529,-32.445,37.304,-179.9898,0.0316,-6228.9437
C01497=93.155,-36.342,37.389,-179.9982,0.0048,-6231.3119
C01498=91.569,-40.172,37.389,-179.9979,0.0047,-6233.6874
C01499=89.784,-43.901,37.304,-179.9849,0.0296,-6236.0569
C01500=87.565,-47.309,37.176,-179.2873,0.8115,-6238.3812
C01501=84.674,-49.784,37.049,-178.8962,0.6847,-6240.4534
C01502=81.641,-50.965,36.894,-177.9329,0.2906,-6241.9748
C01503=78.886,-50.762,36.600,-178.1553,-0.3569,-6242.7607
C01504=76.172,-50.101,36.009,178.7121,0.3392,-6243.3343
C01505=73.649,-49.580,35.239,171.8007,1.3907,-6243.9482
C01506=71.353,-49.662,34.490,159.1242,-2.4573,-6244.8381
C01507=69.025,-50.912,33.943,151.5734,-21.8610,-6246.4120
C01508=66.209,-53.858,33.725,153.8288,-28.9327,-6249.1268
C01509=63.397,-57.102,33.716,153.6142,-28.9918,-6252.0095
C01510=60.334,-60.334,33.722,152.2694,-27.7301,-6255.0000
C01511=57.102,-63.397,33.716,151.0085,-26.3861,-6257.9905
C01512=53.858,-66.209,33.725,151.0682,-26.1719,-6260.8732
C01513=50.912,-69.025,33.943,158.1383,-28.4263,-6263.5880
C01514=49.662,-71.353,34.490,177.5427,-20.8758,-6265.1619
C01515=49.580,-73.649,35.239,-178.6093,-8.1993,-6266.0518
C01516=50.101,-76.172,36.009,-179.6608,-1.2879,-6266.6657
C01517=50.762,-78.886,36.600,179.6431,1.8447,-6267.2393
C01518=50.965,-81.641,36.894,-179.7094,2.0671,-6268.0252
C01519=49.784,-84.674,37.049,-179.3153,1.1038,-6269.5466
C01520=47.309,-87.565,37.176,-179.1885,0.7127,-6271.6188
C01521=43.901,-89.784,37.304,-179.9704,0.0151,-6273.9431
C01522=40.172,-91.569,37.389,-179.9953,0.0021,-6276.3126
C01523=36.342,-93.155,37.389,-179.9952,0.0018,-6278.6881
C01524=32.445,-94.529,37.304,-179.9684,0.0102,-6281.0563
C01525=28.465,-95.370,37.176,-178.9222,0.0699,-6283.3813
C01526=24.671,-95.076,37.049,-178.7354,-0.2964,-6285.4533
C01527=21.692,-93.766,36.894,-178.3326,-1.2566,-6286.9742
C01528=19.887,-91.675,36.600,-178.9476,-1.5568,-6287.7605
C01529=18.435,-89.289,36.009,179.3291,1.1505,-6288.3344
C01530=17.019,-87.137,35.239,175.1574,6.7892,-6288.9485
C01531=15.338,-85.570,34.490,163.2997,13.4594,-6289.8379
C01532=12.808,-84.808,33.943,146.3185,5.6572,-6291.4119
C01533=8.733,-84.900,33.725,143.5590,-2.4835,-6294.1271
C01534=4.451,-85.206,33.716,143.4019,-2.3496,-6297.0097
C01535=0.000,-85.325,33.722,143.3716,0.0004,-6300.0000
C01536=0.000,-85.325,33.722,143.3716,0.0004,-6300.0000
C01537=-4.451,-85.206,33.716,143.4018,2.3490,-6302.9903
C01538=-8.733,-84.900,33.725,143.5591,2.4820,-6305.8729
C01539=-12.808,-84.808,33.943,146.3182,-5.6564,-6308.5881
C01540=-15.338,-85.570,34.490,163.2997,-13.4594,-6310.1621
C01541=-17.019,-87.137,35.239,175.1574,-6.7892,-6311.0515
C01542=-18.435,-89.289,36.009,179.3291,-1.1505,-6311.6656
C01543=-19.887,-91.675,36.600,-178.9476,1.5568,-6312.2395
C01544=-21.692,-93.766,36.894,-178.3326,1.2566,-6313.0258
C01545=-24.671,-95.076,37.049,-178.7354,0.2964,-6314.5467
C01546=-28.465,-95.370,37.176,-178.9222,-0.0699,-6316.6187
C01547=-32.445,-94.529,37.304,-179.9684,-0.0102,-6318.9437
C01548=-36.342,-93.155,37.389,-179.9952,-0.0018,-6321.3119
C01549=-40.172,-91.569,37.389,-179.9953,-0.0021,-6323.6874
C01550=-43.901,-89.784,37.304,-179.9704,-0.0151,-6326.0569
C01551=-47.309,-87.565,37.176,-179.1885,-0.7127,-6328.3812
C01552=-49.784,-84.674,37.049,-179.3153,-1.1038,-6330.4534
C01553=-50.965,-81.641,36.894,-179.7094,-2.0671,-6331.9748
C01554=-50.762,-78.886,36.600,179.6431,-1.8447,-6332.7607
C01555=-50.101,-76.172,36.009,-179.6608,1.2879,-6333.3343
C01556=-49.580,-73.649,35.239,-178.6093,8.1993,-6333.9482
C01557=-49.662,-71.353,34.490,177.5427,20.8758,-6334.8381
C01558=-50.912,-69.025,33.943,158.1390,28.4266,-6336.4120
C01559=-53.858,-66.209,33.725,151.0673,26.1712,-6339.1268
C01560=-57.102,-63.397,33.716,151.0082,26.3858,-6342.0095
C01561=-60.334,-60.334,33.722,152.2699,27.7306,-6345.0000
C01562=-63.397,-57.102,33.716,153.6139,28.9915,-6347.9905
C01563=-66.209,-53.858,33.725,153.8281,28.9318,-6350.8732
C01564=-69.025,-50.912,33.943,151.5737,21.8617,-6353.5880
C01565=-71.353,-49.662,34.490,159.1242,2.4573,-6355.1619
C01566=-73.649,-49.580,35.239,171.8007,-1.3907,-6356.0518
C01567=-76.172,-50.101,36.009,178.7121,-0.3392,-6356.6657
C01568=-78.886,-50.762,36.600,-178.1553,0.3569,-6357.2393
C01569=-81.641,-50.965,36.894,-177.9329,-0.2906,-6358.0252
C01570=-84.674,-49.784,37.049,-178.8962,-0.6847,-6359.5466
C01571=-87.565,-47.309,37.176,-179.2873,-0.8115,-6361.6188
C01572=-89.784,-43.901,37.304,-179.9849,-0.0296,-6363.9431
C01573=-91.569,-40.172,37.389,-179.9979,-0.0047,-6366.3126
C01574=-93.155,-36.342,37.389,-179.9982,-0.0048,-6368.6881
C01575=-94.529,-32.445,37.304,-179.9898,-0.0316,-6371.0563
C01576=-95.370,-28.465,37.176,-179.9301,-1.0778,-6373.3813
C01577=-95.076,-24.671,37.049,179.7036,-1.2646,-6375.4533
C01578=-93.766,-21.692,36.894,178.7434,-1.6674,-6376.9742
C01579=-91.675,-19.887,36.600,178.4432,-1.0524,-6377.7605
C01580=-89.289,-18.435,36.009,-178.8495,0.6709,-6378.3344
C01581=-87.137,-17.019,35.239,-173.2108,4.8426,-6378.9485
C01582=-85.570,-15.338,34.490,-166.5406,16.7003,-6379.8379
C01583=-84.808,-12.808,33.943,-174.3428,33.6815,-6381.4119
C01584=-84.900,-8.733,33.725,177.5165,36.4410,-6384.1271
C01585=-85.206,-4.451,33.716,177.6504,36.5981,-6387.0097
C01586=-85.325,0.000,33.722,-179.9996,36.6284,-6390.0000
C01587=-85.206,4.451,33.716,-177.6510,36.5982,-6392.9903
C01588=-84.900,8.733,33.725,-177.5180,36.4409,-6395.8729
C01589=-84.808,12.808,33.943,174.3436,33.6818,-6398.5881
C01590=-85.570,15.338,34.490,166.5406,16.7003,-6400.1621
C01591=-87.137,17.019,35.239,173.2108,4.8426,-6401.0515
C01592=-89.289,18.435,36.009,178.8495,0.6709,-6401.6656
C01593=-91.675,19.887,36.600,-178.4432,-1.0524,-6402.2395
C01594=-93.766,21.692,36.894,-178.7434,-1.6674,-6403.0258
C01595=-95.076,24.671,37.049,-179.7036,-1.2646,-6404.5467
C01596=-95.370,28.465,37.176,179.9301,-1.0778,-6406.6187
C01597=-94.529,32.445,37.304,179.9898,-0.0316,-6408.9437
C01598=-93.155,36.342,37.389,179.9982,-0.0048,-6411.3119
C01599=-91.569,40.172,37.389,179.9979,-0.0047,-6413.6874
C01600=-89.784,43.901,37.304,179.9849,-0.0296,-6416.0569
C01601=-87.565,47.309,37.176,179.2873,-0.8115,-6418.3812
C01602=-84.674,49.784,37.049,178.8962,-0.6847,-6420.4534
C01603=-81.641,50.965,36.894,177.9329,-0.2906,-6421.9748
C01604=-78.886,50.762,36.600,178.1553,0.3569,-6422.7607
C01605=-76.172,50.101,36.009,-178.7121,-0.3392,-6423.3343
C01606=-73.649,49.580,35.239,-171.8007,-1.3907,-6423.9482
C01607=-71.353,49.662,34.490,-159.1242,2.4573,-6424.8381
C01608=-69.025,50.912,33.943,-151.5734,21.8610,-6426.4120
C01609=-66.209,53.858,33.725,-153.8288,28.9327,-6429.1268
C01610=-63.397,57.102,33.716,-153.6142,28.9918,-6432.0095
C01611=-60.334,60.334,33.722,-152.2694,27.7301,-6435.0000
C01612=-57.102,63.397,33.716,-151.0085,26.3861,-6437.9905
C01613=-53.858,66.209,33.725,-151.0682,26.1719,-6440.8732
C01614=-50.912,69.025,33.943,-158.1383,28.4263,-6443.5880
C01615=-49.662,71.353,34.490,-177.5427,20.8758,-6445.1619
C01616=-49.580,73.649,35.239,178.6093,8.1993,-6446.0518
C01617=-50.101,76.172,36.009,179.6608,1.2879,-6446.6657
C01618=-50.762,78.886,36.600,-179.6431,-1.8447,-6447.2393
C01619=-50.965,81.641,36.894,179.7094,-2.0671,-6448.0252
C01620=-49.784,84.674,37.049,179.3153,-1.1038,-6449.5466
C01621=-47.309,87.565,37.176,179.1885,-0.7127,-6451.6188
C01622=-43.901,89.784,37.304,179.9704,-0.0151,-6453.9431
C01623=-40.172,91.569,37.389,179.9953,-0.0021,-6456.3126
C01624=-36.342,93.155,37.389,179.9952,-0.0018,-6458.6881
C01625=-32.445,94.529,37.304,179.9684,-0.0102,-6461.0563
C01626=-28.465,95.370,37.176,178.9222,-0.0699,-6463.3813
C01627=-24.671,95.076,37.049,178.7354,0.2964,-6465.4533
C01628=-21.692,93.766,36.894,178.3326,1.2566,-6466.9742
C01629=-19.887,91.675,36.600,178.9476,1.5568,-6467.7605
C01630=-18.435,89.289,36.009,-179.3291,-1.1505,-6468.3344
C01631=-17.019,87.137,35.239,-175.1574,-6.7892,-6468.9485
C01632=-15.338,85.570,34.490,-163.2997,-13.4594,-6469.8379
C01633=-12.808,84.808,33.943,-146.3182,-5.6564,-6471.4119
C01634=-8.733,84.900,33.725,-143.5591,2.4820,-6474.1271
C01635=-4.451,85.206,33.716,-143.4018,2.3490,-6477.0097
C01636=0.000,85.325,33.722,-143.3716,0.0004,-6480.0000
C01637=0.000,84.003,35.480,-142.7415,0.0004,-6480.0000
C01638=4.330,83.888,35.473,-142.7716,-2.3891,-6482.9548
C01639=8.530,83.594,35.484,-142.9366,-2.3020,-6485.8263
C01640=12.558,83.543,35.726,-146.1518,6.8812,-6488.5486
C01641=15.030,84.409,36.333,-165.2581,13.5086,-6490.0964
C01642=16.662,86.143,37.169,-176.3239,5.7975,-6490.9471
C01643=18.041,88.518,38.031,-179.9182,0.1571,-6491.5198
C01644=19.458,91.164,38.697,178.4928,-2.5231,-6492.0484
C01645=21.221,93.510,39.027,177.6909,-1.9849,-6492.7860
C01646=24.227,95.023,39.203,178.2776,-0.4750,-6494.3034
C01647=28.112,95.435,39.346,178.7289,0.0594,-6496.4132
C01648=32.220,94.603,39.491,179.9530,0.0151,-6498.8079
C01649=36.266,93.184,39.587,179.9934,0.0025,-6501.2653
C01650=40.247,91.535,39.587,179.9935,0.0029,-6503.7346
C01651=44.111,89.678,39.491,179.9560,0.0226,-6506.1917
C01652=47.604,87.360,39.346,179.0591,0.8569,-6508.5867
C01653=50.060,84.322,39.203,179.1177,1.5538,-6510.6966
C01654=51.116,81.128,39.027,179.7705,3.0349,-6512.2136
C01655=50.704,78.221,38.697,-179.2808,2.8489,-6512.9519
C01656=49.835,75.348,38.031,179.9468,-0.1689,-6513.4806
C01657=49.130,72.694,37.169,178.4898,-6.6859,-6514.0527
C01658=49.058,70.314,36.333,-179.0727,-19.5923,-6514.9034
C01659=50.194,67.954,35.726,-158.7492,-29.2297,-6516.4513
C01660=53.078,65.141,35.484,-150.6424,-26.8233,-6519.1737
C01661=56.256,62.380,35.473,-150.4564,-26.9203,-6522.0450
C01662=59.399,59.399,35.480,-151.7261,-28.2744,-6525.0000
C01663=62.380,56.256,35.473,-153.0793,-29.5434,-6527.9550
C01664=65.141,53.078,35.484,-153.1760,-29.3567,-6530.8263
C01665=67.954,50.194,35.726,-150.7705,-21.2516,-6533.5487
C01666=70.314,49.058,36.333,-160.4077,-0.9273,-6535.0966
C01667=72.694,49.130,37.169,-173.3141,1.5102,-6535.9473
C01668=75.348,49.835,38.031,-179.8311,0.0532,-6536.5194
C01669=78.221,50.704,38.697,177.1511,-0.7192,-6537.0481
C01670=81.128,51.116,39.027,176.9651,0.2295,-6537.7864
C01671=84.322,50.060,39.203,178.4462,0.8823,-6539.3034
C01672=87.360,47.604,39.346,179.1431,0.9409,-6541.4133
C01673=89.678,44.111,39.491,179.9774,0.0440,-6543.8083
C01674=91.535,40.247,39.587,179.9971,0.0065,-6546.2654
C01675=93.184,36.266,39.587,179.9975,0.0066,-6548.7347
C01676=94.603,32.220,39.491,179.9849,0.0470,-6551.1921
C01677=95.435,28.112,39.346,179.9406,1.2711,-6553.5868
C01678=95.023,24.227,39.203,-179.5250,1.7224,-6555.6966
C01679=93.510,21.221,39.027,-178.0151,2.3091,-6557.2140
C01680=91.164,19.458,38.697,-177.4769,1.5072,-6557.9516
C01681=88.518,18.041,38.031,179.8429,-0.0818,-6558.4802
C01682=86.143,16.662,37.169,174.2025,-3.6761,-6559.0529
C01683=84.409,15.030,36.333,166.4914,-14.7419,-6559.9036
C01684=83.543,12.558,35.726,173.1188,-33.8482,-6561.4514
C01685=83.594,8.530,35.484,-177.6980,-37.0634,-6564.1737
C01686=83.888,4.330,35.473,-177.6109,-37.2284,-6567.0452
C01687=84.003,0.000,35.480,179.9996,-37.2585,-6570.0000
C01688=83.888,-4.330,35.473,177.6115,-37.2285,-6572.9548
C01689=83.594,-8.530,35.484,177.6995,-37.0633,-6575.8263
C01690=83.543,-12.558,35.726,-173.1197,-33.8485,-6578.5486
C01691=84.409,-15.030,36.333,-166.4914,-14.7419,-6580.0964
C01692=86.143,-16.662,37.169,-174.2025,-3.6761,-6580.9471
C01693=88.518,-18.041,38.031,-179.8429,-0.0818,-6581.5198
C01694=91.164,-19.458,38.697,177.4769,1.5072,-6582.0484
C01695=93.510,-21.221,39.027,178.0151,2.3091,-6582.7860
C01696=95.023,-24.227,39.203,179.5250,1.7224,-6584.3034
C01697=95.435,-28.112,39.346,-179.9406,1.2711,-6586.4132
C01698=94.603,-32.220,39.491,-179.9849,0.0470,-6588.8079
C01699=93.184,-36.266,39.587,-179.9975,0.0066,-6591.2653
C01700=91.535,-40.247,39.587,-179.9971,0.0065,-6593.7346
C01701=89.678,-44.111,39.491,-179.9774,0.0440,-6596.1917
C01702=87.360,-47.604,39.346,-179.1431,0.9409,-6598.5867
C01703=84.322,-50.060,39.203,-178.4462,0.8823,-6600.6966
C01704=81.128,-51.116,39.027,-176.9651,0.2295,-6602.2136
C01705=78.221,-50.704,38.697,-177.1511,-0.7192,-6602.9519
C01706=75.348,-49.835,38.031,179.8311,0.0532,-6603.4806
C01707=72.694,-49.130,37.169,173.3141,1.5102,-6604.0527
C01708=70.314,-49.058,36.333,160.4077,-0.9273,-6604.9034
C01709=67.954,-50.194,35.726,150.7703,-21.2508,-6606.4513
C01710=65.141,-53.078,35.484,153.1767,-29.3576,-6609.1737
C01711=62.380,-56.256,35.473,153.0797,-29.5436,-6612.0450
C01712=59.399,-59.399,35.480,151.7256,-28.2739,-6615.0000
C01713=56.256,-62.380,35.473,150.4566,-26.9207,-6617.9550
C01714=53.078,-65.141,35.484,150.6433,-26.8240,-6620.8263
C01715=50.194,-67.954,35.726,158.7484,-29.2295,-6623.5487
C01716=49.058,-70.314,36.333,179.0727,-19.5923,-6625.0966
C01717=49.130,-72.694,37.169,-178.4898,-6.6859,-6625.9473
C01718=49.835,-75.348,38.031,-179.9468,-0.1689,-6626.5194
C01719=50.704,-78.221,38.697,179.2808,2.8489,-6627.0481
C01720=51.116,-81.128,39.027,-179.7705,3.0349,-6627.7864
C01721=50.060,-84.322,39.203,-179.1177,1.5538,-6629.3034
C01722=47.604,-87.360,39.346,-179.0591,0.8569,-6631.4133
C01723=44.111,-89.678,39.491,-179.9560,0.0226,-6633.8083
C01724=40.247,-91.535,39.587,-179.9935,0.0029,-6636.2654
C01725=36.266,-93.184,39.587,-179.9934,0.0025,-6638.7347
C01726=32.220,-94.603,39.491,-179.9530,0.0151,-6641.1921
C01727=28.112,-95.435,39.346,-178.7289,0.0594,-6643.5868
C01728=24.227,-95.023,39.203,-178.2776,-0.4750,-6645.6966
C01729=21.221,-93.510,39.027,-177.6909,-1.9849,-6647.2140
C01730=19.458,-91.164,38.697,-178.4928,-2.5231,-6647.9516
C01731=18.041,-88.518,38.031,179.9182,0.1571,-6648.4802
C01732=16.662,-86.143,37.169,176.3239,5.7975,-6649.0529
C01733=15.030,-84.409,36.333,165.2581,13.5086,-6649.9036
C01734=12.558,-83.543,35.726,146.1518,6.8812,-6651.4514
C01735=8.530,-83.594,35.484,142.9366,-2.3020,-6654.1737
C01736=4.330,-83.888,35.473,142.7716,-2.3891,-6657.0452
C01737=0.000,-84.003,35.480,142.7415,0.0004,-6660.0000
C01738=0.000,-84.003,35.480,142.7415,0.0004,-6660.0000
C01739=-4.330,-83.888,35.473,142.7715,2.3885,-6662.9548
C01740=-8.530,-83.594,35.484,142.9367,2.3005,-6665.8263
C01741=-12.558,-83.543,35.726,146.1515,-6.8803,-6668.5486
C01742=-15.030,-84.409,36.333,165.2581,-13.5086,-6670.0964
